// TIA Portal project "Factory IO Linha Completa" (V18)

(* hardware
DEVICE "S7-1500/ET200MP station_1"  S7-1500 station
   slot 0: "Rail_0"  Rack  6ES7 590-1***0-0AA0
   slot 1: "PLC_1"  CPU 1515-2 PN  6ES7 515-2AM00-0AB0  V1.8
      slot 3: "CPU display_1"  6ES7591-1BA00-0AA0
      slot 32768: "PROFINET interface_1"  X1
         slot 32769: "Port_1"  X1 P1
         slot 32770: "Port_2"  X1 P2
      slot 33024: "PROFINET interface_2"  X2
         slot 33025: "Port_1"  X2 P1
*)

// ===== PLC "PLC_1"  CPU 1515-2 PN =====

VAR_GLOBAL   // PLC tag table "Default tag table"
   "System_Byte" AT %MB1 : Byte;
   "FirstScan" AT %M1.0 : Bool;
   "DiagStatusUpdate" AT %M1.1 : Bool;
   "AlwaysTRUE" AT %M1.2 : Bool;
   "AlwaysFALSE" AT %M1.3 : Bool;
   "Clock_Byte" AT %MB0 : Byte;
   "Clock_10Hz" AT %M0.0 : Bool;
   "Clock_5Hz" AT %M0.1 : Bool;
   "Clock_2.5Hz" AT %M0.2 : Bool;
   "Clock_2Hz" AT %M0.3 : Bool;
   "Clock_1.25Hz" AT %M0.4 : Bool;
   "Clock_1Hz" AT %M0.5 : Bool;
   "Clock_0.625Hz" AT %M0.6 : Bool;
   "Clock_0.5Hz" AT %M0.7 : Bool;
END_VAR

VAR_GLOBAL   // PLC tag table "FactoryIO"
   "Emergency Stop 0" AT %I0.0 : Bool;
   "Start Button 0" AT %I0.1 : Bool;
   "Stop Button 0" AT %I0.2 : Bool;
   "Reset Button 0" AT %I0.3 : Bool;
   "Machining Center 0 (Is Busy)" AT %I0.5 : Bool;
   "Machining Center 0 (Has Error)" AT %I0.6 : Bool;
   "Machining Center 1 (Is Busy)" AT %I0.7 : Bool;
   "Machining Center 1 (Has Error)" AT %I1.0 : Bool;
   "Sensor 120" AT %I1.1 : Bool;
   "Sensor 122" AT %I1.2 : Bool;
   "Zne01 Conveyor 101" AT %Q0.0 : Bool;
   "Zne01 Conveyor 120" AT %Q0.1 : Bool;
   "Zne01 Conveyor 121" AT %Q0.2 : Bool;
   "Zne01 Conveyor 122" AT %Q0.3 : Bool;
   "Zne01 Conveyor 124" AT %Q0.4 : Bool;
   "Zne01 Conveyor 125" AT %Q0.5 : Bool;
   "Zne01 Sorter 102 (Up)" AT %Q0.6 : Bool;
   "Zne01 Sorter 102 (Left)" AT %Q0.7 : Bool;
   "Zne01 Sorter 102 (Right)" AT %Q1.0 : Bool;
   "Zne01 Sorter 123 (Up)" AT %Q1.1 : Bool;
   "Zne01 Sorter 123 (Right)" AT %Q1.2 : Bool;
   "Machining Center 0 (Start)" AT %Q1.3 : Bool;
   "Machining Center 0 (Stop)" AT %Q1.4 : Bool;
   "Machining Center 0 (Reset)" AT %Q1.5 : Bool;
   "Machining Center 1 (Start)" AT %Q1.6 : Bool;
   "Machining Center 1 (Stop)" AT %Q1.7 : Bool;
   "Machining Center 1 (Reset)" AT %Q2.0 : Bool;
   "Start Button 0 (Light)" AT %Q2.1 : Bool;
   "Stop Button 0 (Light)" AT %Q2.2 : Bool;
   "Reset Button 0 (Light)" AT %Q2.3 : Bool;
   "Vision Sensor 0 (Value)" AT %IW256 : Int;
   "Auto Selector 0" AT %I0.4 : Bool;
   "Machining Center 2 (Is Busy)" AT %I1.3 : Bool;
   "Machining Center 2 (Has Error)" AT %I1.4 : Bool;
   "Machining Center 3 (Is Busy)" AT %I1.5 : Bool;
   "Machining Center 3 (Has Error)" AT %I1.6 : Bool;
   "Sensor 130" AT %I1.7 : Bool;
   "Sensor 132" AT %I2.0 : Bool;
   "Zne01 Conveyor 130" AT %Q2.4 : Bool;
   "Zne01 Conveyor 131" AT %Q2.5 : Bool;
   "Zne01 Conveyor 132" AT %Q2.6 : Bool;
   "Zne01 Conveyor 134" AT %Q2.7 : Bool;
   "Zne01 Conveyor 135" AT %Q3.0 : Bool;
   "Zne01 Sorter 133 (Up)" AT %Q3.1 : Bool;
   "Zne01 Sorter 133 (Left)" AT %Q3.2 : Bool;
   "Machining Center 2 (Start)" AT %Q3.3 : Bool;
   "Machining Center 2 (Stop)" AT %Q3.4 : Bool;
   "Machining Center 2 (Reset)" AT %Q3.5 : Bool;
   "Machining Center 3 (Start)" AT %Q3.6 : Bool;
   "Machining Center 3 (Stop)" AT %Q3.7 : Bool;
   "Machining Center 3 (Reset)" AT %Q4.0 : Bool;
   "Zne02 Conveyor 220" AT %Q4.1 : Bool;
   "Zne02 Conveyor 221" AT %Q4.2 : Bool;
   "Zne02 Conveyor 222A" AT %Q4.3 : Bool;
   "Zne02 Conveyor 222B" AT %Q4.4 : Bool;
   "Zne02 Conveyor 223" AT %Q4.5 : Bool;
   "Zne02 Conveyor 224" AT %Q4.6 : Bool;
   "Zne02 Conveyor 225" AT %Q4.7 : Bool;
   "Zne03 Conveyor 300" AT %Q5.3 : Bool;
   "Zne03 Conveyor 301" AT %Q5.4 : Bool;
   "Zne03 Conveyor 302" AT %Q5.5 : Bool;
   "Sensor 223" AT %I2.1 : Bool;
   "Sensor 225" AT %I2.2 : Bool;
   "Zne02 Clamp Closed" AT %I2.3 : Bool;
   "Zne02 Clamp Limit" AT %I2.4 : Bool;
   "Zne02 Pusher" AT %Q5.0 : Bool;
   "Zne02 Clamp" AT %Q5.1 : Bool;
   "Zne02 Clamp Rise" AT %Q5.2 : Bool;
   "Vision Sensor 2 (Value)" AT %IW258 : Int;
   "Sensor 300" AT %I2.5 : Bool;
   "Sensor 301" AT %I2.6 : Bool;
   "Sensor 302" AT %I2.7 : Bool;
   "Zne03 (Detected)" AT %I3.0 : Bool;
   "Zne03 (Moving X)" AT %I3.1 : Bool;
   "Zne03 (Moving Z)" AT %I3.2 : Bool;
   "Zne03 Clamp Closed" AT %I3.3 : Bool;
   "Zne03 Clamp Limit" AT %I3.4 : Bool;
   "Zne03 Clamp" AT %Q5.6 : Bool;
   "Zne03 Clamp Raise" AT %Q5.7 : Bool;
   "Zne03 X" AT %Q6.0 : Bool;
   "Zne03 Z" AT %Q6.1 : Bool;
   "Zne03 (Grab)" AT %Q6.2 : Bool;
   "Zne03 Pusher" AT %Q6.3 : Bool;
   "Vision Sensor 1 (Value)" AT %IW260 : Int;
   "Sensor 423" AT %I3.5 : Bool;
   "Sensor 425" AT %I3.6 : Bool;
   "Zne04 Clamp Closed" AT %I3.7 : Bool;
   "Zne04 Clamp Limit" AT %I4.0 : Bool;
   "Sensor 500" AT %I4.1 : Bool;
   "Sensor 501" AT %I4.2 : Bool;
   "Sensor 502" AT %I4.3 : Bool;
   "Zne05 (Detected)" AT %I4.4 : Bool;
   "Zne05 (Moving X)" AT %I4.5 : Bool;
   "Zne05 (Moving Z)" AT %I4.6 : Bool;
   "Zne05 Clamp Closed" AT %I4.7 : Bool;
   "Zne05 Clamp Limit" AT %I5.0 : Bool;
   "Zne04 Conveyor 420" AT %Q6.4 : Bool;
   "Zne04 Conveyor 421" AT %Q6.5 : Bool;
   "Zne04 Conveyor 422B" AT %Q6.7 : Bool;
   "Zne04 Conveyor 423" AT %Q7.0 : Bool;
   "Zne04 Conveyor 424" AT %Q7.1 : Bool;
   "Zne04 Conveyor 425" AT %Q7.2 : Bool;
   "Zne04 Pusher" AT %Q7.3 : Bool;
   "Zne04 Clamp" AT %Q7.4 : Bool;
   "Zne04 Clamp Raise" AT %Q7.5 : Bool;
   "Zne05 Conveyor 500" AT %Q7.6 : Bool;
   "Zne05 Conveyor 501" AT %Q7.7 : Bool;
   "Zne05 Conveyor 502" AT %Q8.0 : Bool;
   "Zne05 Clamp" AT %Q8.1 : Bool;
   "Zne05 Clamp Raise" AT %Q8.2 : Bool;
   "Zne05 X" AT %Q8.3 : Bool;
   "Zne05 Z" AT %Q8.4 : Bool;
   "Zne05 (Grab)" AT %Q8.5 : Bool;
   "Zne05 Pusher" AT %Q8.6 : Bool;
   "Vision Sensor 3 (Value)" AT %IW262 : Int;
   "Vision Sensor 4 (Value)" AT %IW264 : Int;
   "Zne04 Conveyor 422A" AT %Q6.6 : Bool;
   "Sensor 920" AT %I10.0 : Bool;
   "Sensor 921" AT %I10.1 : Bool;
   "Sensor 922" AT %I10.2 : Bool;
   "Sensor 930" AT %I10.3 : Bool;
   "Sensor 931" AT %I10.4 : Bool;
   "Sensor 932" AT %I10.5 : Bool;
   "Sensor 950" AT %I10.6 : Bool;
   "Sensor 951" AT %I10.7 : Bool;
   "Sensor 952" AT %I11.0 : Bool;
   "Sensor 953" AT %I11.1 : Bool;
   "Zne09 Conveyor 920" AT %Q10.0 : Bool;
   "Zne09 Conveyor 921" AT %Q10.1 : Bool;
   "Zne09 Conveyor 930" AT %Q10.2 : Bool;
   "Zne09 Conveyor 931" AT %Q10.3 : Bool;
   "Zne09 Conveyor 950" AT %Q10.4 : Bool;
   "Zne09 Conveyor 951" AT %Q10.5 : Bool;
   "Zne09 Conveyor 952" AT %Q10.6 : Bool;
   "Zne09 Conveyor 953" AT %Q10.7 : Bool;
   "Zne09 Chain Transfer Right" AT %Q11.0 : Bool;
   "Zne09 Chain Transfer Left" AT %Q11.1 : Bool;
   "Zne09 Chain Transfer Foward" AT %Q11.2 : Bool;
   "Zne09 Chain Transfer Backward" AT %Q11.3 : Bool;
   "Pick & Place 0 X Position (V)" AT %IW266 : Int;
   "Pick & Place 0 Y Position (V)" AT %IW268 : Int;
   "Pick & Place 0 Z Position (V)" AT %IW270 : Int;
   "Pick & Place 1 X Position (V)" AT %IW272 : Int;
   "Pick & Place 1 Y Position (V)" AT %IW274 : Int;
   "Pick & Place 1 Z Position (V)" AT %IW276 : Int;
   "Pick & Place 0 X Set Point (V)" AT %QW256 : Int;
   "Pick & Place 0 Y Set Point(V)" AT %QW258 : Int;
   "Pick & Place 0 Z Set Point (V)" AT %QW260 : Int;
   "Pick & Place 1 X Set Point (V)" AT %QW262 : Int;
   "Pick & Place 1 Y Set Point(V)" AT %QW264 : Int;
   "Pick & Place 1 Z Set Point (V)" AT %QW266 : Int;
   "Zne09 Stacker Target Position" AT %QW270 : Int;
   "Pick & Place 1 (Box Detected)" AT %I11.2 : Bool;
   "Pick & Place 0 (Box Detected)" AT %I11.3 : Bool;
   "Pick & Place 1 (Grab)" AT %Q11.4 : Bool;
   "Pick & Place 0 (Grab)" AT %Q11.5 : Bool;
   "AtRight" AT %I12.0 : Bool;
   "AtLeft" AT %I12.1 : Bool;
   "AtCenter" AT %I12.2 : Bool;
   "MovingX" AT %I12.3 : Bool;
   "MovingZ" AT %I12.4 : Bool;
   "Forks RIght" AT %Q12.0 : Bool;
   "ForksLeft" AT %Q12.1 : Bool;
   "Lift" AT %Q12.2 : Bool;
END_VAR

VAR_GLOBAL CONSTANT   // PLC tag table "FactoryIO"
   "BlueRawMaterial" : Int := 1;
   "GreenRawMaterial" : Int := 4;
   "HOMEPOSITION" : Int := 255;
   "BlueLidMaterial" : Int := 2;
   "GreenLidMaterial" : Int := 5;
   "BlueBaseMaterial" : Int := 3;
   "GreenBaseMaterial" : Int := 6;
   "MaxCoordinates" : Int := 10;
END_VAR

TYPE "St_Conveyor"
   STRUCT
      IHM_xButtonRun : Bool;
      IHM_xStatusMotor : Int;
      iq_xError : Bool;
      iq_iErrorType : Int;
   END_STRUCT;
END_TYPE

TYPE "St_ControlPanel"
   STRUCT
      q_xManualMode : Bool;
      q_xAutoMode : Bool;
      q_xEmergencyStatusZone : Bool;
      q_xPanelResetCmd : Bool;
      iq_xPanelOn : Bool;
      iq_xPanelOff : Bool;
      iq_xError : Bool;
      iq_iErrorType : Int;
      q_siMode : Int;
      iq_sFaultDescription : String;
   END_STRUCT;
END_TYPE

TYPE "St_Warehouse"
   STRUCT
      xPedidoRetirada : Bool;
      xFimMovimento : Bool;
      xPosiçaoLivre : Bool;
      iPosição : Int;
      xSensorEntrada : Bool;
      xSensorSaida : Bool;
      iMachineState_Entrada : Int;
      iMachineState_Retirada : Int;
      xForksLeft : Bool;
      xForksRight : Bool;
      xLift : Bool;
      q_dTargetPosition : DInt;
      Armazem : Array[1..54] of Bool;
      iStateRetirada : String;
      iStateEntrada : String;
   END_STRUCT;
END_TYPE

TYPE "St_Sorter"
   STRUCT
      temp : Bool;
   END_STRUCT;
END_TYPE

TYPE "St_Assembler"
   STRUCT
      LidClampUpPosition : Bool;
      LidClampDownPosition : Bool;
      BaseClampUpPosition : Bool;
      BaseClampDownPosition : Bool;
      AxisXFoward : Bool;
      AxisXBackward : Bool;
      AxisZRise : Bool;
      AxisZDown : Bool;
      iMachineState : Int;
      iState : String;
      MemoryPresenceLid : Bool;
      MemoryPresenceBase : Bool;
      ReadyToReceiveLid : Bool;
      ReadyToReceiveBase : Bool;
      EnableSend : Bool;
   END_STRUCT;
END_TYPE

TYPE "St_Manipulator"
   STRUCT
      ReadyToReceivePallet : Bool;
      PalletFull : Bool;
      ContActual : Int;
      ContMax : Int;
      iMachineState : Int;
      iState : String;
      Coordinates : Array[0.."MaxCoordinates"] of Struct
         "Axis X" : Int;
         "Axis Y" : Int;
         "Axis Z" : Int;
      END_STRUCT;
      Ack_Positions : Array[0.."MaxCoordinates"] of Bool;
   END_STRUCT;
END_TYPE

TYPE "St_Transfer"
   STRUCT
      EnableSend : Bool;
      RequestRight : Bool;
      RequestLeft : Bool;
      ReadyToReceiveRight : Bool;
      ReadyToReceiveLeft : Bool;
      LastReceiveRightSide : Bool;
      "Chain Transfer Foward" : Bool;
      "Chain Transfer Backward" : Bool;
      "Chain Transfer Right" : Bool;
      "Chain Transfer Left" : Bool;
      iMachineState : Int;
      iState : String;
   END_STRUCT;
END_TYPE

DATA_BLOCK "General"   // DB2
{ S7_Optimized_Access := 'TRUE' }
VERSION : 0.1
   VAR
      Panel01 : "St_ControlPanel";
      "Conveyor 101" : "St_Conveyor";
      "Conveyor 120" : "St_Conveyor";
      "Conveyor 121" : "St_Conveyor";
      "Conveyor 122" : "St_Conveyor";
      "Conveyor 124" : "St_Conveyor";
      "Conveyor 125" : "St_Conveyor";
      "Conveyor 130" : "St_Conveyor";
      "Conveyor 131" : "St_Conveyor";
      "Conveyor 132" : "St_Conveyor";
      "Conveyor 134" : "St_Conveyor";
      "Conveyor 135" : "St_Conveyor";
      "Conveyor 220" : "St_Conveyor";
      "Conveyor 221" : "St_Conveyor";
      "Conveyor 222" : "St_Conveyor";
      "Conveyor 223" : "St_Conveyor";
      "Conveyor 224" : "St_Conveyor";
      "Conveyor 225" : "St_Conveyor";
      "Conveyor 300" : "St_Conveyor";
      "Conveyor 301" : "St_Conveyor";
      "Conveyor 302" : "St_Conveyor";
      "Assembler Zne03" : "St_Assembler";
      "Conveyor 420" : "St_Conveyor";
      "Conveyor 421" : "St_Conveyor";
      "Conveyor 422" : "St_Conveyor";
      "Conveyor 423" : "St_Conveyor";
      "Conveyor 424" : "St_Conveyor";
      "Conveyor 425" : "St_Conveyor";
      "Conveyor 500" : "St_Conveyor";
      "Conveyor 501" : "St_Conveyor";
      "Conveyor 502" : "St_Conveyor";
      "Assembler Zne05" : "St_Assembler";
      "Conveyor 920" : "St_Conveyor";
      "Conveyor 921" : "St_Conveyor";
      "Manipulator 1" : "St_Manipulator";
      "Conveyor 930" : "St_Conveyor";
      "Conveyor 931" : "St_Conveyor";
      "Manipulator 0" : "St_Manipulator";
      Transfer : "St_Transfer";
      "Conveyor 950" : "St_Conveyor";
      "Conveyor 951" : "St_Conveyor";
      Warehouse : "St_Warehouse";
      "Conveyor 952" : "St_Conveyor";
      "Conveyor 953" : "St_Conveyor";
   END_VAR
BEGIN
END_DATA_BLOCK

// folder: PANEL

DATA_BLOCK "ControlPanel_DB"   // DB1
{ S7_Optimized_Access := 'TRUE' }
VERSION : 0.1
// stored: InstanceOfName ControlPanel
"ControlPanel"
BEGIN
END_DATA_BLOCK

// folder: ZNE01

DATA_BLOCK "Zne01_DB"   // DB3
{ S7_Optimized_Access := 'TRUE' }
VERSION : 0.1
// stored: InstanceOfName Zne01
"Zne01"
BEGIN
END_DATA_BLOCK

// folder: ZNE02

DATA_BLOCK "Zne02_DB"   // DB4
{ S7_Optimized_Access := 'TRUE' }
VERSION : 0.1
// stored: InstanceOfName Zne02
"Zne02"
BEGIN
END_DATA_BLOCK

// folder: ZNE03

DATA_BLOCK "Zne03_DB"   // DB5
{ S7_Optimized_Access := 'TRUE' }
VERSION : 0.1
// stored: InstanceOfName Zne03
"Zne03"
BEGIN
END_DATA_BLOCK

// folder: ZNE04

DATA_BLOCK "Zne04_DB"   // DB6
{ S7_Optimized_Access := 'TRUE' }
VERSION : 0.1
// stored: InstanceOfName Zne04
"Zne04"
BEGIN
END_DATA_BLOCK

// folder: ZNE05

DATA_BLOCK "Zne05_DB"   // DB7
{ S7_Optimized_Access := 'TRUE' }
VERSION : 0.1
// stored: InstanceOfName Zne05
"Zne05"
BEGIN
END_DATA_BLOCK

// folder: ZNE09

DATA_BLOCK "Zne09_DB"   // DB8
{ S7_Optimized_Access := 'TRUE' }
VERSION : 0.1
// stored: InstanceOfName Zne09
"Zne09"
BEGIN
END_DATA_BLOCK

// folder: (top level)

ORGANIZATION_BLOCK "Main_1"   // OB123, SCL, ProgramCycle
TITLE = "Main Program Sweep (Cycle)"
{ S7_Optimized_Access := 'TRUE' }
VERSION : 0.1
   VAR_INPUT
      Initial_Call : Bool;   // Initial call of this OB
      Remanence : Bool;   // =True, if remanent data are available
   END_VAR
BEGIN


   "MHJ-PLC-Lab-Function-S71200"();

   "ControlPanel_DB"(i_xButtonReset:="Reset Button 0",
                     i_xButtonStart:="Start Button 0",
                     i_xButtonStop:="Stop Button 0",
                     i_xButtonEmergency:="Emergency Stop 0",
                     i_xSelectorMode:="Auto Selector 0",
                     i_xClock:="Clock_1Hz",
                     q_xStartLight=>"Start Button 0 (Light)",
                     q_xStopLight=>"Stop Button 0 (Light)",
                     q_xResetLight=>"Reset Button 0 (Light)",
                     ControlPanel:="General".Panel01);

   "Zne01_DB"(); 
   "Zne02_DB"();
   "Zne03_DB"();
   "Zne04_DB"();
   "Zne05_DB"();
   "Receita"();
   "Zne09_DB"();
END_ORGANIZATION_BLOCK

// folder: PANEL

FUNCTION_BLOCK "ControlPanel"   // FB1, SCL
{ S7_Optimized_Access := 'TRUE' }
VERSION : 0.1
   VAR_INPUT
      i_xButtonReset : Bool;
      i_xButtonStart : Bool;
      i_xButtonStop : Bool;
      i_xButtonEmergency : Bool;
      i_xSelectorMode : Bool;   // 0 = Manual, 1= Auto
      i_xClock : Bool;
   END_VAR
   VAR_OUTPUT
      q_xStartLight : Bool;
      q_xStopLight : Bool;
      q_xResetLight : Bool;
   END_VAR
   VAR_IN_OUT
      ControlPanel : "St_ControlPanel";
   END_VAR
   VAR
      IEC_Timer_0_Instance : TON_TIME;
   END_VAR
BEGIN
   REGION INPUTS
       //EMERGENCY STATUS//
       IF #i_xButtonEmergency AND #i_xButtonReset THEN
           #ControlPanel.q_xEmergencyStatusZone := TRUE;
       ELSIF NOT #i_xButtonEmergency THEN
           #ControlPanel.q_xEmergencyStatusZone := FALSE;
       END_IF;

       //MANUAL MODE//
       IF #ControlPanel.q_xEmergencyStatusZone AND NOT #i_xSelectorMode THEN
           #ControlPanel.q_xManualMode := TRUE;
       ELSIF NOT #ControlPanel.q_xEmergencyStatusZone OR #i_xSelectorMode THEN
           #ControlPanel.q_xManualMode := FALSE;
       END_IF;

       //AUTO MODE//
       IF #ControlPanel.q_xEmergencyStatusZone AND #i_xSelectorMode AND #ControlPanel.iq_xPanelOn THEN
           #ControlPanel.q_xAutoMode := TRUE;
       ELSIF NOT #ControlPanel.q_xEmergencyStatusZone OR NOT #i_xSelectorMode OR #ControlPanel.iq_xPanelOff THEN
           #ControlPanel.q_xAutoMode := FALSE;
       END_IF;

       //RESET COMMAND//
       #IEC_Timer_0_Instance(IN:=#i_xButtonReset,
                             PT:=t#5s,
                             Q=>#ControlPanel.q_xPanelResetCmd);

       //ON-OFF COMMAND//
       IF #i_xButtonStart AND #i_xButtonStop THEN
           #ControlPanel.iq_xPanelOn := TRUE;
           #ControlPanel.iq_xPanelOff := FALSE;
       ELSIF NOT #i_xButtonStop OR NOT #ControlPanel.q_xEmergencyStatusZone OR #ControlPanel.q_xManualMode THEN
           #ControlPanel.iq_xPanelOn := FALSE;
           #ControlPanel.iq_xPanelOff := TRUE;
       END_IF;
   END_REGION

   REGION STATUS MODE
       IF NOT #ControlPanel.q_xEmergencyStatusZone THEN
           #ControlPanel.q_siMode := 1; //EMERGENCIA

       ELSIF #ControlPanel.q_xAutoMode THEN
           #ControlPanel.q_siMode := 2; //AUTOMATICO

       ELSIF #ControlPanel.q_xManualMode THEN
           #ControlPanel.q_siMode := 3; //MANUAL

       ELSE
           #ControlPanel.q_siMode := 4; //DESLIGADO
       END_IF;
   END_REGION

   REGION OUTPUTS
       //START LIGHT    
       #q_xStartLight := #ControlPanel.q_xAutoMode OR (#i_xSelectorMode AND #ControlPanel.q_xEmergencyStatusZone AND #i_xClock);
       //STOP LIGHT 
       #q_xStopLight := NOT #i_xButtonEmergency OR (#i_xButtonEmergency AND NOT #ControlPanel.q_xEmergencyStatusZone AND #i_xClock);
       //RESET LIGHT 
       #q_xResetLight := #ControlPanel.q_xPanelResetCmd;
   END_REGION
END_FUNCTION_BLOCK

// folder: STANDARD BLOCKS

FUNCTION_BLOCK "Conveyor"   // FB2, SCL
{ S7_Optimized_Access := 'TRUE' }
VERSION : 0.1
   VAR_INPUT
      i_xInterlock : Bool;
      i_xRun : Bool;
      ControlPanel : "St_ControlPanel";
   END_VAR
   VAR_OUTPUT
      q_xMotorOn : Bool := false;
   END_VAR
   VAR_IN_OUT
      Conveyor : "St_Conveyor";
   END_VAR
BEGIN

   REGION MODO
       CASE #ControlPanel.q_siMode OF
           1:  // EMERGENCIA
               #q_xMotorOn := FALSE;

           2:  // AUTOMATICO
               IF #i_xRun AND NOT #i_xInterlock THEN
                   #q_xMotorOn := TRUE;
               ELSE
                   #q_xMotorOn := FALSE;
               END_IF;

           3:  // MANUAL
               #q_xMotorOn := #Conveyor.IHM_xButtonRun;

           ELSE
               #q_xMotorOn := FALSE;
       END_CASE;
   END_REGION

   REGION #IHM
       IF #Conveyor.iq_xError THEN
           #Conveyor.IHM_xStatusMotor := 1; // ERRO

       ELSIF #ControlPanel.q_xAutoMode AND #q_xMotorOn THEN
           #Conveyor.IHM_xStatusMotor := 2; // AUTO RUNNING

       ELSIF #ControlPanel.q_xManualMode AND #q_xMotorOn THEN
           #Conveyor.IHM_xStatusMotor := 3; // MANUAL RUNNING

       ELSIF NOT #q_xMotorOn THEN
           #Conveyor.IHM_xStatusMotor := 4; // MOTOR STOPED

       END_IF;
   END_REGION
END_FUNCTION_BLOCK

FUNCTION_BLOCK "Warehouse"   // FB3, SCL
{ S7_Optimized_Access := 'TRUE' }
VERSION : 0.1
   VAR_INPUT
      i_xAtLeft : Bool;
      i_xAtRight : Bool;
      i_xAtMiddle : Bool;
      i_xMovingZ : Bool;
      i_xMovingX : Bool;
      ControlPanel : "St_ControlPanel";
   END_VAR
   VAR_OUTPUT
      q_xForksLeft : Bool;
      q_xForksRight : Bool;
      q_xLift : Bool;
      q_dTargetPosition : Int;
   END_VAR
   VAR_IN_OUT
      Warehouse : "St_Warehouse";
   END_VAR
   VAR
      t_LiftDown : TON_TIME;
      t_LiftUp : TON_TIME;
      TargetPositionRetirada : DInt;
      TargetPositionEntrada : DInt;
      t_NotMovingX : TON_TIME;
   END_VAR
BEGIN

   IF #ControlPanel.q_xPanelResetCmd THEN
       #Warehouse.xForksLeft := 0;
       #Warehouse.xForksRight := 0;
       #Warehouse.xLift := 0;
       #Warehouse.q_dTargetPosition := "HOMEPOSITION";
       #Warehouse.iMachineState_Entrada := 0;
       #Warehouse.iMachineState_Retirada := 0;
       #Warehouse.iPosição := 0;
   END_IF;


   IF #Warehouse.iPosição > 54 THEN
       #Warehouse.iPosição := 54;
   END_IF;

   IF #Warehouse.iPosição < 1 THEN
       #Warehouse.iPosição := 1;
   END_IF;

   REGION TIMMERS
       #t_LiftDown(IN := NOT #q_xLift AND NOT #i_xMovingZ,
                   PT := T#1s);

       #t_LiftUp(IN:=#q_xLift AND NOT #i_xMovingZ,
                 PT:=T#1s);

       #t_NotMovingX(IN:= NOT #i_xMovingX,
                  PT:=T#2s);
   END_REGION

   REGION ESTADO RETIRADA
       IF #ControlPanel.q_xAutoMode AND #Warehouse.iMachineState_Entrada <= 1 THEN

           CASE #Warehouse.iMachineState_Retirada OF
               0:  // AGUARDANDO SOLICITAÇÃO RETIRADA
                   #Warehouse.iStateRetirada := 'S00 - AGUARDANDO SOLICITACAO RETIRADA';
                   IF #Warehouse.xPedidoRetirada THEN
                       #Warehouse.iMachineState_Retirada := 1;
                   END_IF;

               1:  // VERIFICA POSICAO VALIDA
                   #Warehouse.iStateRetirada := 'S01 - VERIFICA POSICAO VALIDA';
                   IF #Warehouse.Armazem[#Warehouse.iPosição] THEN
                       #Warehouse.iMachineState_Retirada := 3;
                       #TargetPositionRetirada := #Warehouse.iPosição;
                   ELSE
                       #Warehouse.iMachineState_Retirada := 2;
                   END_IF;

               2:  // POSICAO INVALIDA
                   #Warehouse.iStateRetirada := 'S02 - POSICAO INVALIDA PARA RETIRADA';
                   IF NOT #Warehouse.xPedidoRetirada THEN
                       #Warehouse.iMachineState_Retirada := 0;
                   END_IF;

               3:  // FORK LIVRE
                   #Warehouse.iStateRetirada := 'S03 - REPOUSO FORKS';
                   #Warehouse.xLift := 0;
                   IF #t_LiftDown.Q THEN
                       #Warehouse.xForksLeft := 0;
                       #Warehouse.xForksRight := 0;
                       IF #i_xAtMiddle THEN
                           #Warehouse.iMachineState_Retirada := 4;
                       END_IF;
                   END_IF;

               4:  // DESLOCA PARA POSICAO DO ARMAZEM
                   #Warehouse.iStateRetirada := 'S04 - DESLOCA PARA POSICAO DO ARMAZEM';
                   #Warehouse.q_dTargetPosition := #TargetPositionRetirada;
                   IF (#q_dTargetPosition = #Warehouse.q_dTargetPosition) AND #t_NotMovingX.Q THEN
                       #Warehouse.iMachineState_Retirada := 5;
                   END_IF;

               5:  // AVANCA FORK
                   #Warehouse.iStateRetirada := 'S05 - AVANCA FORK';
                   #Warehouse.xForksRight := 1;
                   IF #q_xForksRight AND #i_xAtRight THEN
                       #Warehouse.iMachineState_Retirada := 6;
                   END_IF;

               6:  // LIFT UP
                   #Warehouse.iStateRetirada := 'S06 - ERGUE LIFT';
                   #Warehouse.xLift := 1;
                   IF #q_xLift AND #t_LiftUp.Q THEN
                       #Warehouse.Armazem[#TargetPositionRetirada] := 0;
                       IF NOT #Warehouse.Armazem[#TargetPositionRetirada] THEN
                           #Warehouse.iMachineState_Retirada := 7;
                       END_IF;
                   END_IF;

               7:  // RECUA FORKS
                   #Warehouse.iStateRetirada := 'S07 - RECUA FORKS';
                   #Warehouse.xForksRight := 0;
                   IF NOT #q_xForksRight AND #i_xAtMiddle THEN
                       #Warehouse.iMachineState_Retirada := 8;
                   END_IF;

               8:  // DESLOCA PARA POSICAO DAS ESTEIRA DE SAIDA
                   #Warehouse.iStateRetirada := 'S08 - DESLOCA PARA POSICAO DAS ESTEIRA DE SAIDA';
                   #Warehouse.q_dTargetPosition := "HOMEPOSITION";
                   IF #t_NotMovingX.Q AND (#q_dTargetPosition = "HOMEPOSITION") AND NOT #Warehouse.xSensorSaida THEN
                       #Warehouse.iMachineState_Retirada := 9;
                   END_IF;

               9:  // AVANCA FORK PARA ENVIO ESTEIRA
                   #Warehouse.iStateRetirada := 'S09 - AVANCA FORK PARA ENVIO ESTEIRA';
                   #Warehouse.xForksRight := 1;
                   IF #q_xForksRight AND #i_xAtRight THEN
                       #Warehouse.iMachineState_Retirada := 10;
                   END_IF;

               10: // LIFT DOWN
                   #Warehouse.iStateRetirada := 'S10 - DEPOSITA PALLET NA ESTEIRA';
                   #Warehouse.xLift := 0;
                   IF NOT #q_xLift AND #t_LiftDown.Q THEN
                       #Warehouse.iMachineState_Retirada := 11;
                   END_IF;

               11: // RECUA FORKS
                   #Warehouse.iStateRetirada := 'S11 - RECUA FORKS';
                   #Warehouse.xForksRight := 0;
                   IF NOT #q_xForksRight AND #i_xAtMiddle AND NOT #Warehouse.xPedidoRetirada THEN
                       #Warehouse.iMachineState_Retirada := 0;
                       #Warehouse.iStateRetirada := 'S00 - AGUARDANDO SOLICITACAO RETIRADA';
                   END_IF;

               ELSE
                   #Warehouse.iMachineState_Retirada := 0;
           END_CASE;
       END_IF;
   END_REGION

   REGION ESTADO DEPOSITO 

       IF #ControlPanel.q_xAutoMode AND #Warehouse.iMachineState_Retirada = 0 THEN

           CASE #Warehouse.iMachineState_Entrada OF

               0: //POSICAO LIVRE INDISPONIVEL
                   #Warehouse.iStateEntrada := 'S00 - POSICAO LIVRE INDISPONIVEL';
                   #TargetPositionEntrada := "PosDisponivel"(#Warehouse.Armazem);
                   IF #TargetPositionEntrada <> -1 THEN
                       #Warehouse.iMachineState_Entrada := 1;
                   END_IF;

               1:  // AGUARDANDO CHEGADA PALLET
                   #Warehouse.iStateEntrada := 'S01 - AGUARDANDO CHEGADA PALLET';
                   IF #Warehouse.xSensorEntrada AND NOT #Warehouse.xPedidoRetirada THEN
                       #Warehouse.iMachineState_Entrada := 2;
                   END_IF;

               2:   // VERIFICA POSICAO DISPONIVEL
                   #Warehouse.iStateEntrada := 'S02 - VERIFICA POSICAO DISPONIVEL';
                   #TargetPositionEntrada := "PosDisponivel"(#Warehouse.Armazem);
                   IF #TargetPositionEntrada = -1 THEN
                       #Warehouse.iMachineState_Entrada := 0;
                   ELSE
                       #Warehouse.iMachineState_Entrada := 3;
                   END_IF;

               3: // FORKS LIVRE
                   #Warehouse.iStateEntrada := 'S03 - REPOUSO FORKS';
                   #Warehouse.xLift := 0;
                   IF #t_LiftDown.Q THEN
                       #Warehouse.xForksLeft := 0;
                       #Warehouse.xForksRight := 0;
                       IF #i_xAtMiddle THEN
                           #Warehouse.iMachineState_Entrada := 4;
                       END_IF;
                   END_IF;

               4: // DESLOCA PARA POSICAO DA ESTEIRA DE ENTRADA
                   #Warehouse.iStateEntrada := 'S04 - DESLOCA PARA POSICAO DA ESTEIRA DE ENTRADA';
                   #Warehouse.q_dTargetPosition := "HOMEPOSITION";
                   IF #q_dTargetPosition = "HOMEPOSITION" AND #t_NotMovingX.Q THEN
                       #Warehouse.iMachineState_Entrada := 5;
                   END_IF;

               5: // AVANÇA FORKS
                   #Warehouse.iStateEntrada := 'S05 - AVANCA FORKS';
                   #Warehouse.xForksLeft := 1;
                   IF #q_xForksLeft AND #i_xAtLeft THEN
                       #Warehouse.iMachineState_Entrada := 6;
                   END_IF;

               6:  // RETIRAR PALLET
                   #Warehouse.iStateEntrada := 'S06 - RETIRAR PALLET';
                   #Warehouse.xLift := 1;
                   IF #q_xLift AND #t_LiftUp.Q AND NOT #Warehouse.xSensorEntrada THEN
                       #Warehouse.iMachineState_Entrada := 7;
                   END_IF;

               7: // RECUA FORKS
                   #Warehouse.iStateEntrada := 'S07 - RECUA FORKS';
                   #Warehouse.xForksLeft := 0;
                   IF NOT #Warehouse.xForksLeft AND #i_xAtMiddle THEN
                       #Warehouse.iMachineState_Entrada := 8;
                   END_IF;

               8: // DESLOCA PARA POSICAO DE DEPOSITO NO ARMAZEM
                   #Warehouse.iStateEntrada := 'S08 - DESLOCA PARA POSICAO DE DEPOSITO NO ARMAZEM';
                   #Warehouse.q_dTargetPosition := #TargetPositionEntrada;
                   IF #q_dTargetPosition = #TargetPositionEntrada AND #t_NotMovingX.Q THEN
                       #Warehouse.iMachineState_Entrada := 9;
                   END_IF;

               9: // AVANÇA FORKS NO ARMAZEM
                   #Warehouse.iStateEntrada := 'S09 - AVANCA FORKS NO ARMAZEM';
                   #Warehouse.xForksRight := 1;
                   IF #q_xForksRight AND #i_xAtRight THEN
                       #Warehouse.iMachineState_Entrada := 10;
                   END_IF;

               10: // DEPOSITA PALLET
                   #Warehouse.iStateEntrada := 'S10 - DEPOSITA PALLET';
                   #Warehouse.xLift := 0;
                   IF NOT #q_xLift AND #t_LiftDown.Q THEN
                       #Warehouse.Armazem[#q_dTargetPosition] := 1;
                       #Warehouse.iMachineState_Entrada := 11;
                   END_IF;

               11: // RECUA FORKS
                   #Warehouse.iStateEntrada := 'S11 - RECUA FORKS APOS DEPOSITO';
                   #Warehouse.xForksRight := 0;
                   IF NOT #q_xForksRight AND #i_xAtMiddle THEN
                       #Warehouse.iMachineState_Entrada := 0;
                   END_IF;

               ELSE  
                   #Warehouse.iMachineState_Entrada := 0;
           END_CASE;
       END_IF;
   END_REGION




   REGION OUTPUTS
       IF #ControlPanel.q_xAutoMode THEN

           IF #t_NotMovingX.Q THEN 
               #q_xForksLeft := #Warehouse.xForksLeft;
               #q_xForksRight := #Warehouse.xForksRight;
               #q_xLift := #Warehouse.xLift;
           END_IF;

           IF #i_xAtMiddle AND NOT #q_xForksLeft AND NOT #q_xForksRight THEN 
               #q_dTargetPosition := #Warehouse.q_dTargetPosition;
           END_IF;

       END_IF;
   END_REGION
END_FUNCTION_BLOCK

FUNCTION_BLOCK "Sorter"   // FB5, SCL
{ S7_Optimized_Access := 'TRUE' }
VERSION : 0.1
   VAR_INPUT
      i_xRightRequest : Bool;
      i_xLeftRequest : Bool;
      i_xCenterRequest : Bool;
      ControlPanel : "St_ControlPanel";
   END_VAR
   VAR_OUTPUT
      q_xUp : Bool;
      q_xRight : Bool;
      q_xLeft : Bool;
   END_VAR
BEGIN

   REGION MODO
       CASE #ControlPanel.q_siMode OF
           1:  // EMERGENCIA
               #q_xUp := FALSE;

           2:  // AUTOMATICO
               #q_xUp := TRUE;

               IF #i_xRightRequest THEN
                   #q_xRight := TRUE;
                   #q_xLeft := FALSE;
               END_IF;

               IF #i_xLeftRequest THEN
                   #q_xRight := FALSE;
                   #q_xLeft := TRUE;
               END_IF;

               IF #i_xCenterRequest THEN
                   #q_xRight := FALSE;
                   #q_xLeft := FALSE;
               END_IF;

           3:  // MANUAL
               #q_xUp := FALSE;

           ELSE
               #q_xUp := FALSE;
       END_CASE;
   END_REGION
END_FUNCTION_BLOCK

FUNCTION_BLOCK "MachineCenter"   // FB6, SCL
{ S7_Optimized_Access := 'TRUE' }
VERSION : 0.1
   VAR_INPUT
      Interlock : Bool;
      ControlPanel : "St_ControlPanel";
   END_VAR
   VAR_OUTPUT
      Start : Bool;
      Stop : Bool;
      Reset : Bool;
   END_VAR
BEGIN
   REGION MODO
       CASE #ControlPanel.q_siMode OF
           1:  // EMERGENCIA
               #Start := FALSE;
               #Stop := TRUE;

           2:  // AUTOMATICO
               IF NOT #Interlock THEN
                   #Start := TRUE;
                   #Stop := FALSE;
               ELSE
                   #Start := FALSE;
                   #Stop := TRUE;
               END_IF;

           3:  // MANUAL
               #Start := FALSE;
               #Stop := TRUE;

           ELSE
               #Start := FALSE;
               #Stop := TRUE;
       END_CASE;
   END_REGION

   #Reset := #ControlPanel.q_xPanelResetCmd;
END_FUNCTION_BLOCK

FUNCTION_BLOCK "Pusher"   // FB8, SCL
{ S7_Optimized_Access := 'TRUE' }
VERSION : 0.1
   VAR_INPUT
      RequestPusher : Bool;
      "Timer" : Time;
      ControlPanel : "St_ControlPanel";
   END_VAR
   VAR_OUTPUT
      Pusher : Bool;
   END_VAR
   VAR
      RequestPusherDelay : TON_TIME;
   END_VAR
BEGIN

   REGION MODO
       CASE #ControlPanel.q_siMode OF
           1:  // EMERGENCIA
               #Pusher := FALSE;

           2:  // AUTOMATICO
               #RequestPusherDelay(IN:=#RequestPusher,
                                   PT:=#Timer);

               IF #RequestPusherDelay.Q THEN
                   #Pusher := TRUE;
               ELSE
                   #Pusher := FALSE;
               END_IF;

           3:  // MANUAL
               #Pusher := FALSE;

           ELSE
               #Pusher := FALSE;
       END_CASE;
   END_REGION
END_FUNCTION_BLOCK

FUNCTION_BLOCK "Assembler"   // FB10, SCL
{ S7_Optimized_Access := 'TRUE' }
VERSION : 0.1
   VAR_INPUT
      LidClampClosed : Bool;
      LidClampLimit : Bool;
      BaseClampClosed : Bool;
      BaseClampLimit : Bool;
      PresenceLidConveyor : Bool;
      PresenceBaseConveyor : Bool;
      PresenceGrab : Bool;
      MovingX : Bool;
      MovingZ : Bool;
      ControlPanel : "St_ControlPanel";
   END_VAR
   VAR_OUTPUT
      LidClampClose : Bool;
      LidClampRise : Bool;
      BaseClampClose : Bool;
      BaseClampRise : Bool;
      AxisX : Bool;
      AxisZ : Bool;
      Grab : Bool;
   END_VAR
   VAR_IN_OUT
      "St_ Assembler" : "St_Assembler";
   END_VAR
   VAR
      iMachineState : Int;
      LidPresence : F_TRIG;
      BasePresence : F_TRIG;
      tVacuoOff : TON_TIME;
      tSaidaPeça : TON_TIME;
      tLidClampUp : TON_TIME;
      tLidClampDown : TON_TIME;
      tBaseClampUp : TON_TIME;
      tBaseClampDown : TON_TIME;
      tXFoward : TON_TIME;
      tXBackward : TON_TIME;
      tZRise : TON_TIME;
      tZDown : TON_TIME;
   END_VAR
BEGIN
   REGION Memory Presence
       #LidPresence(CLK := #PresenceLidConveyor); // PULSE LID PRESENCE
       IF #LidPresence.Q THEN
           #"St_ Assembler".MemoryPresenceLid := 1;
       END_IF;

       #BasePresence(CLK := #PresenceBaseConveyor); // PULSE BASE PRESENCE
       IF #BasePresence.Q THEN
           #"St_ Assembler".MemoryPresenceBase := 1;
       END_IF;
   END_REGION

   REGION HOME MACHINE
       IF #ControlPanel.q_xPanelResetCmd THEN
           #LidClampClose := 0;
           #LidClampRise := 0;
           #BaseClampClose := 0;
           #BaseClampRise := 0;
           #AxisX := 1;
           #AxisZ := 0;
           #Grab := 0;
           #"St_ Assembler".iMachineState := 0;
           #"St_ Assembler".MemoryPresenceLid := 0;
           #"St_ Assembler".MemoryPresenceBase := 0;
       END_IF;
   END_REGION

   REGION Timmers
       #tVacuoOff(IN := NOT #Grab,
                  PT := T#500ms);

       #tSaidaPeça(IN:=#BaseClampRise,
                   PT:=T#3s);

       #tLidClampUp(IN:=#LidClampRise AND #LidClampLimit ,
                    PT:=T#300ms,
                    Q=>#"St_ Assembler".LidClampUpPosition);

       #tLidClampDown(IN:=NOT #LidClampRise AND #LidClampLimit,
                      PT:=T#300ms,
                      Q=>#"St_ Assembler".LidClampDownPosition);

       #tBaseClampUp(IN:=#BaseClampRise AND #BaseClampLimit,
                     PT:=T#300ms,
                     Q=>#"St_ Assembler".BaseClampUpPosition);

       #tBaseClampDown(IN:=NOT #BaseClampRise AND #BaseClampLimit,
                       PT:=T#300ms,
                       Q=>#"St_ Assembler".BaseClampDownPosition);

       #tXFoward(IN:=#AxisX AND NOT #MovingX ,
                 PT:=T#300ms,
                 Q=>#"St_ Assembler".AxisXFoward);

       #tXBackward(IN:= NOT #AxisX AND NOT #MovingX,
                   PT:=T#300ms,
                   Q=>#"St_ Assembler".AxisXBackward);

       #tZRise(IN:=NOT #AxisZ AND NOT #MovingZ,
               PT:=T#300ms,
               Q=>#"St_ Assembler".AxisZRise);

       #tZDown(IN:=#AxisZ AND NOT #MovingZ,
               PT:=T#300ms,
               Q=>#"St_ Assembler".AxisZDown);
   END_REGION

   // READY TO RECEIVE SIGNAL
   #"St_ Assembler".ReadyToReceiveLid := #ControlPanel.q_xAutoMode AND #"St_ Assembler".iMachineState = 1 AND NOT #"St_ Assembler".MemoryPresenceLid;
   #"St_ Assembler".ReadyToReceiveBase := #ControlPanel.q_xAutoMode AND #"St_ Assembler".iMachineState = 1 AND NOT #"St_ Assembler".MemoryPresenceBase;
   IF #ControlPanel.q_xAutoMode THEN
       CASE #"St_ Assembler".iMachineState OF
           0:  // HOME MACHINE
               #"St_ Assembler".iState := 'S00 PASSO INICIAL';
               #LidClampClose := FALSE;
               #LidClampRise := FALSE;
               #BaseClampClose := FALSE;
               #BaseClampRise := FALSE;
               #AxisX := TRUE;
               #AxisZ := FALSE;
               #Grab := FALSE;

               IF NOT #LidClampClosed AND #"St_ Assembler".LidClampDownPosition AND NOT #BaseClampClosed AND #"St_ Assembler".BaseClampDownPosition AND #"St_ Assembler".AxisXFoward AND #"St_ Assembler".AxisZRise THEN
                   #"St_ Assembler".iMachineState := 1;
               END_IF;
               ;
           1:  // AGUARDANDO LID E BASE PRESENÇA
               #"St_ Assembler".iState := 'S01 AGUARDANDO LID E BASE PRESENCA';
               IF #"St_ Assembler".MemoryPresenceLid THEN
                   #LidClampClose := 1;
               END_IF;
               IF #"St_ Assembler".MemoryPresenceBase THEN
                   #BaseClampClose := 1;
               END_IF;
               IF #LidClampClosed AND #BaseClampClosed AND #"St_ Assembler".MemoryPresenceBase AND #"St_ Assembler".MemoryPresenceLid THEN
                   #"St_ Assembler".iMachineState := 2;
               END_IF;

           2: // PICK POSITION
               #"St_ Assembler".iState := 'S02 PICK POSITION';
               #AxisX := 1;
               IF #"St_ Assembler".AxisXFoward THEN
                   #AxisZ := 1;
               END_IF;
               IF #"St_ Assembler".AxisXFoward AND #"St_ Assembler".AxisZDown THEN
                   #"St_ Assembler".iMachineState := 3;
               END_IF;

           3: // ACIONA VACUO
               #"St_ Assembler".iState := 'S03 ACIONA VACUO';
               #Grab := 1;
               IF #Grab AND #PresenceGrab THEN
                   #"St_ Assembler".iMachineState := 4;
               END_IF;

           4: // RETIRA LID 
               #"St_ Assembler".iState := 'S04 RETIRA LID';
               #LidClampClose := 0;
               #AxisZ := 0;
               IF NOT #LidClampClosed AND #"St_ Assembler".AxisZRise AND #PresenceGrab THEN
                   #"St_ Assembler".MemoryPresenceLid := 0;
                   #"St_ Assembler".iMachineState := 5;
               END_IF;

           5: // RECUA EIXO X
               #"St_ Assembler".iState := 'S05 RECUA EIXO X';
               #AxisX := 0;
               IF #"St_ Assembler".AxisXBackward THEN
                   #"St_ Assembler".iMachineState := 6;
               END_IF;

           6: // DESCE PARA MONTAGEM
               #"St_ Assembler".iState := 'S06 DESCE PARA MONTAGEM';
               #AxisZ := 1;
               IF #"St_ Assembler".AxisZDown THEN
                   #"St_ Assembler".iMachineState := 7;
               END_IF;

           7: // LIBERA VACUO
               #"St_ Assembler".iState := 'S07 LIBERA VACUO';
               #Grab := 0;
               IF #tVacuoOff.Q THEN
                   #"St_ Assembler".iMachineState := 8;
               END_IF;

           8: // SOBE SEM PEÇA
               #"St_ Assembler".iState := 'S08 SOBE SEM PECA';
               #AxisZ := 0;
               #BaseClampClose := 0;
               IF NOT #BaseClampClosed AND #"St_ Assembler".AxisZRise AND NOT #PresenceGrab AND #"St_ Assembler".EnableSend THEN
                   #"St_ Assembler".iMachineState := 9;
               END_IF;

           9: // LIBERA PEÇA COMPLETA
               #"St_ Assembler".iState := 'S09 LIBERA PECA COMPLETA';
               #AxisX := 1;
               #BaseClampRise := 1;
               IF #"St_ Assembler".AxisXFoward AND #tSaidaPeça.Q THEN
                   #"St_ Assembler".MemoryPresenceBase := 0;
                   #"St_ Assembler".iMachineState := 0;
               END_IF;
           ELSE  
               #"St_ Assembler".iMachineState := 0; 
       END_CASE;
   END_IF;
END_FUNCTION_BLOCK

FUNCTION_BLOCK "Manipulator"   // FB14, SCL
{ S7_Optimized_Access := 'TRUE' }
VERSION : 0.1
   VAR_INPUT
      "Pallet Detected" : Bool;
      "Part Detected" : Bool;
      PresenceGrab : Bool;
      "Actual Position X" : Int;
      "Actual Position Y" : Int;
      "Actual Position Z" : Int;
      ControlPanel : "St_ControlPanel";
   END_VAR
   VAR_OUTPUT
      "X Setpoint" : Int;
      "Y Setpoint" : Int;
      "Z Setpoint" : Int;
      Grab : Bool;
   END_VAR
   VAR_IN_OUT
      Manipulator : "St_Manipulator";
   END_VAR
   VAR
      Position : Struct
         x : Int;
         y : Int;
         z : Int;
      END_STRUCT;
      "Null Position" : Bool;
      i : Int;
      GrabOff : TON_TIME;
      NotPallet : TON_TIME;
   END_VAR
   VAR CONSTANT
      Tolerance : Int := 30;
      Offset : Int := -2000;
   END_VAR
   // // Manipulator.Coordinates[0] : Home
   // // Manipulator.Coordinates[1] : PrePick
   // // Manipulator.Coordinates[2] : Pick
   // // Manipulator.Coordinates[3] : PosPick
   // // Manipulator.Coordinates[4] : PreDrop
   // // Manipulator.Coordinates[5] : Drop
   // // Manipulator.Coordinates[6] : PosDrop
   // // Manipulator.Ack_Positions[0] : Home
   // // Manipulator.Ack_Positions[1] : PrePick
   // // Manipulator.Ack_Positions[2] : Pick
   // // Manipulator.Ack_Positions[3] : PosPick
   // // Manipulator.Ack_Positions[4] : PreDrop
   // // Manipulator.Ack_Positions[5] : Drop
   // // Manipulator.Ack_Positions[6] : PosDrop
BEGIN

   REGION "General" Reset
       IF #ControlPanel.q_xPanelResetCmd THEN
           #Position := #Manipulator.Coordinates[0]; //Home
           #Grab := 0;
           #Manipulator.ReadyToReceivePallet := 0;
           #Manipulator.PalletFull := 0;
           #Manipulator.ContActual := 0;
           #Manipulator.iMachineState := 0;
       END_IF;

   END_REGION

   REGION Timers
       #GrabOff(IN:=NOT #Grab, PT:=T#1s);
       #NotPallet(IN:=NOT #"Pallet Detected", PT:=T#2s);
   END_REGION

   REGION Acknowledged Position      
       // "General".Manipulator.Coordinates[5]."Axis Z" := 27648 - (#Manipulator.ContActual * 2000);
       FOR #i := 0 TO "MaxCoordinates" DO
           #Manipulator.Ack_Positions[#i] := "Ack Position"("Actual Position X" := #"Actual Position X",
                                                            "Actual Position Y" := #"Actual Position Y",
                                                            "Actual Position Z" := #"Actual Position Z",
                                                            Position := #Manipulator.Coordinates[#i]);
       END_FOR;
   END_REGION

   REGION Machine State
       IF #ControlPanel.q_xAutoMode THEN

           CASE #Manipulator.iMachineState OF
               0:  // RESET CONTADOR
                   #Manipulator.iState := 'S00 PASSO INICIAL';
                   #Manipulator.ContActual := 0;
                   #Manipulator.ReadyToReceivePallet := 0;
                   #Manipulator.PalletFull := 0;
                   IF #Manipulator.ContActual = 0 THEN
                       #Manipulator.iMachineState := 1;
                   END_IF;

               1: // HOME MACHINE 
                   #Manipulator.iState := 'S01 POSICAO INICIAL';
                       #Position := #Manipulator.Coordinates[0];
                       #Grab := 0;
                       IF #Manipulator.Ack_Positions[0] AND NOT #PresenceGrab THEN
                       #Manipulator.iMachineState := 2;
                   END_IF;

               2: // AGUARDANDO PALET E PEÇA
                   #Manipulator.iState := 'S02 AGUARDANDO PALET E PEÇA';
                   #Manipulator.ReadyToReceivePallet := 1;

                   IF #"Pallet Detected" THEN
                       #Manipulator.ReadyToReceivePallet := 0;    
                   END_IF;

                   IF #"Pallet Detected" AND #"Part Detected" THEN
                       #Manipulator.iMachineState := 3;
                       #Manipulator.ReadyToReceivePallet := 0;
                   END_IF;

               3: // PREPICK POSITION
                   #Manipulator.iState := 'S03 PREPICK POSITION';
                   #Position := #Manipulator.Coordinates[1];
                   IF #Manipulator.Ack_Positions[1] THEN
                       #Manipulator.iMachineState := 4;
                   END_IF;

               4: // PICK POSITION
                   #Manipulator.iState := 'S04 PICK POSITION';
                   #Position := #Manipulator.Coordinates[2];
                   IF #Manipulator.Ack_Positions[2] THEN
                       #Manipulator.iMachineState := 5;
                   END_IF;

               5: // LIGAR VACUO 
                   #Manipulator.iState := 'S05 LIGAR VACUO';
                   #Grab := 1;
                   IF #Grab AND #PresenceGrab THEN
                       #Manipulator.iMachineState := 6;
                   END_IF;

               6: // POSPICK POSITION
                   #Manipulator.iState := 'S06 POSPICK POSITION';
                   #Position := #Manipulator.Coordinates[3];
                   IF #Manipulator.Ack_Positions[3] AND #PresenceGrab THEN
                       #Manipulator.iMachineState := 7;
                   END_IF;

               7: //PREDROP POSITION
                   #Manipulator.iState := 'S07 PREDROP POSITION';
                   #Position := #Manipulator.Coordinates[4];
                   IF #Manipulator.Ack_Positions[4] AND #"Pallet Detected" THEN
                       #Manipulator.iMachineState := 8;
                   END_IF;

               8: //DROP POSITION
                   #Manipulator.iState := 'S08 DROP POSITION';
                   #Position := #Manipulator.Coordinates[5];
                   IF #Manipulator.Ack_Positions[5] THEN
                       #Manipulator.iMachineState := 9;
                   END_IF;

               9: // LIBERA VACUO
                   #Manipulator.iState := 'S09 LIBERA VACUO';
                   #Grab := 0;
                   IF #GrabOff.Q THEN
                       #Manipulator.iMachineState := 10;
                   END_IF;

               10: // POS DROP
                   #Manipulator.iState := 'S10 POS DROP';
                   #Position := #Manipulator.Coordinates[6];
                   IF #Manipulator.Ack_Positions[6] AND NOT #PresenceGrab THEN
                       #Manipulator.ContActual := #Manipulator.ContActual + 1;
                       #Manipulator.iMachineState := 11;
                   END_IF;

               11: // VERIFICA CONTADOR
                   #Manipulator.iState := 'S11 VERIFICA CONTADOR';
                   IF #Manipulator.ContActual >= #Manipulator.ContMax THEN

                       #Manipulator.iMachineState := 12;
                   ELSE
                       #Manipulator.iMachineState := 1;
                   END_IF;

               12: //PALET CHEIO
                   #Manipulator.iState := 'S12 PALET CHEIO';
                   #Manipulator.PalletFull := 1;
                   IF #NotPallet.Q THEN
                       #Manipulator.iMachineState := 0;
                   END_IF;
               ELSE  
                   #Manipulator.iMachineState := 0;
           END_CASE;
       END_IF;
   END_REGION

   REGION OFFSET FROP


   END_REGION


   REGION OUTPUTS
       #"X Setpoint" := #Position.x;
       #"Y Setpoint" := #Position.y;
       #"Z Setpoint" := #Position.z;
   END_REGION
END_FUNCTION_BLOCK

FUNCTION_BLOCK "Transfer"   // FB15, SCL
{ S7_Optimized_Access := 'TRUE' }
VERSION : 0.1
   VAR_INPUT
      RightStop : Bool;
      LeftStop : Bool;
      ControlPanel : "St_ControlPanel";
   END_VAR
   VAR_OUTPUT
      "Chain Transfer Foward" : Bool;
      "Chain Transfer Backward" : Bool;
      "Chain Transfer Right" : Bool;
      "Chain Transfer Left" : Bool;
   END_VAR
   VAR_IN_OUT
      Transfer : "St_Transfer";
   END_VAR
BEGIN

   REGION Reset    
       IF #ControlPanel.q_xPanelResetCmd THEN
           #Transfer.iMachineState := 0;
           #Transfer."Chain Transfer Foward" := 0;
           #Transfer."Chain Transfer Backward" := 0;
           #Transfer."Chain Transfer Right" := 0;
           #Transfer."Chain Transfer Left" := 0;
           #Transfer.ReadyToReceiveRight := 0;
           #Transfer.ReadyToReceiveLeft := 0;
       END_IF;
   END_REGION


   REGION Machine State    
       IF #ControlPanel.q_xAutoMode THEN
           CASE #Transfer.iMachineState OF
               0:  // HOME 
                   #Transfer.iState := 'S00 HOME POSITION';
                   #Transfer."Chain Transfer Foward" := 0;
                   #Transfer."Chain Transfer Backward" := 0;
                   #Transfer."Chain Transfer Right" := 0;
                   #Transfer."Chain Transfer Left" := 0;
                   #Transfer.ReadyToReceiveRight := 0;
                   #Transfer.ReadyToReceiveLeft := 0;

                   IF NOT #RightStop AND NOT #LeftStop THEN
                       #Transfer.iMachineState := 1;
                   END_IF;

               1:  // AGUARDA PALET
                   #Transfer.iState := 'S01 AGUARDA PALET';

                   IF #Transfer.RequestRight AND NOT #Transfer.RequestLeft THEN
                       #Transfer.iMachineState := 2;
                   ELSIF NOT #Transfer.RequestRight AND #Transfer.RequestLeft THEN
                       #Transfer.iMachineState := 3;
                   ELSIF #Transfer.RequestRight AND #Transfer.RequestLeft THEN
                       IF #Transfer.LastReceiveRightSide THEN
                           #Transfer.iMachineState := 3;
                       ELSE
                           #Transfer.iMachineState := 2;
                       END_IF;
                   END_IF;

               2: // RECEBE PALET PELA DIREITA
                   #Transfer.iState := 'S02 RECEBE PALET PELA DIREITA';
                   #Transfer.ReadyToReceiveRight := 1;
                   #Transfer."Chain Transfer Right" := 1;
                   IF #RightStop THEN
                       #Transfer.iMachineState := 4;
                       #Transfer.LastReceiveRightSide := 1;
                   END_IF;

               3: // RECEBE PALET PELA ESQUERDA
                   #Transfer.iState := 'S03 RECEBE PALET PELA ESQUERDA';
                   #Transfer.ReadyToReceiveLeft := 1;
                   #Transfer."Chain Transfer Left" := 1;
                   IF #LeftStop THEN
                       #Transfer.iMachineState := 4;
                       #Transfer.LastReceiveRightSide := 0;
                   END_IF;

               4: // AGUARDA LIBERACAO PARA ENVIAR
                   #Transfer.iState := 'S04 AGUARDA LIBERACAO PARA ENVIAR';
                   #Transfer.ReadyToReceiveLeft := 0;
                   #Transfer.ReadyToReceiveRight := 0;
                   #Transfer."Chain Transfer Right" := 0;
                   #Transfer."Chain Transfer Left" := 0;
                   IF #Transfer.EnableSend THEN
                       #Transfer.iMachineState := 5;
                   END_IF;

               5: // ENVIAR PALET 
                   #Transfer.iState := 'S05 AGUARDA LIBERACAO PARA ENVIAR';
                   #Transfer."Chain Transfer Foward" := 1;
                   IF NOT #Transfer.EnableSend THEN
                       #Transfer.iMachineState := 0;
                   END_IF;

               ELSE
                   #Transfer.iMachineState := 0;
           END_CASE;
       END_IF;
   END_REGION

   REGION OUTPUTS
       CASE #ControlPanel.q_siMode OF
           1:  // EMERGENCIA
               #"Chain Transfer Foward" := 0;
               #"Chain Transfer Backward" := 0;
               #"Chain Transfer Right" := 0;
               #"Chain Transfer Left" := 0;

           2:  // AUTOMATICO
               #"Chain Transfer Foward" := #Transfer."Chain Transfer Foward";
               #"Chain Transfer Backward" := #Transfer."Chain Transfer Backward";
               #"Chain Transfer Right" := #Transfer."Chain Transfer Right";
               #"Chain Transfer Left" := #Transfer."Chain Transfer Left";

           3:  // MANUAL
               #"Chain Transfer Foward" := 0;
               #"Chain Transfer Backward" := 0;
               #"Chain Transfer Right" := 0;
               #"Chain Transfer Left" := 0;

           ELSE
               #"Chain Transfer Foward" := 0;
               #"Chain Transfer Backward" := 0;
               #"Chain Transfer Right" := 0;
               #"Chain Transfer Left" := 0;
       END_CASE;
   END_REGION
END_FUNCTION_BLOCK

FUNCTION "PosDisponivel" : DInt   // FC1, SCL
{ S7_Optimized_Access := 'TRUE' }
VERSION : 0.1
   VAR_INPUT
      Armazem : Array[1..54] of Bool;
   END_VAR
   VAR_TEMP
      i : Int;
      j : Int;
      "Array" : Array[1..54] of Int;
   END_VAR
   VAR CONSTANT
      Inicio : Int := 1;
      Fim : Int := 54;
   END_VAR
BEGIN
   //INICIALIZA VARIAVEL
   #PosDisponivel := -1;

   //PRIORIDADE ABASTECIMENTO
   #Array[1] := 1;
   #Array[2] := 10;
   #Array[3] := 19;
   #Array[4] := 28;
   #Array[5] := 37;
   #Array[6] := 46;

   #Array[7] := 2;
   #Array[8] := 11;
   #Array[9] := 20;
   #Array[10] := 29;
   #Array[11] := 38;
   #Array[12] := 47;

   #Array[13] := 3;
   #Array[14] := 12;
   #Array[15] := 21;
   #Array[16] := 30;
   #Array[17] := 39;
   #Array[18] := 48;

   #Array[19] := 4;
   #Array[20] := 13;
   #Array[21] := 22;
   #Array[22] := 31;
   #Array[23] := 40;
   #Array[24] := 49;

   #Array[25] := 5;
   #Array[26] := 14;
   #Array[27] := 23;
   #Array[28] := 32;
   #Array[29] := 41;
   #Array[30] := 50;

   #Array[31] := 6;
   #Array[32] := 15;
   #Array[33] := 24;
   #Array[34] := 33;
   #Array[35] := 42;
   #Array[36] := 51;

   #Array[37] := 7;
   #Array[38] := 16;
   #Array[39] := 25;
   #Array[40] := 34;
   #Array[41] := 43;
   #Array[42] := 52;

   #Array[43] := 8;
   #Array[44] := 17;
   #Array[45] := 26;
   #Array[46] := 35;
   #Array[47] := 44;
   #Array[48] := 53;

   #Array[49] := 9;
   #Array[50] := 18;
   #Array[51] := 27;
   #Array[52] := 36;
   #Array[53] := 45;
   #Array[54] := 54;

   //PROCURA POSICAO LIVRE
   FOR #i := #Inicio TO #Fim DO
       #j := #Array[#i];
       IF NOT #Armazem[#j] THEN
           #PosDisponivel := INT_TO_DINT(#j);
           EXIT;
       END_IF;
   END_FOR;
END_FUNCTION

FUNCTION "Ack Position" : Bool   // FC2, SCL
{ S7_Optimized_Access := 'TRUE' }
VERSION : 0.1
   VAR_INPUT
      "Actual Position X" : Int;
      "Actual Position Y" : Int;
      "Actual Position Z" : Int;
      Position : Struct
         x : Int;
         y : Int;
         z : Int;
      END_STRUCT;
   END_VAR
   VAR_TEMP
      Null : Bool;
   END_VAR
   VAR CONSTANT
      Tolerance : Int := 30;
   END_VAR
BEGIN

   #Null := #"Actual Position X" = 0 OR #"Actual Position Y" = 0 OR #"Actual Position Z" = 0;

   #"Ack Position" := NOT #Null

   AND #"Actual Position X" >= #Position.x - #Tolerance AND #"Actual Position X" <= #Position.x + #Tolerance
   AND #"Actual Position Y" >= #Position.y - #Tolerance AND #"Actual Position Y" <= #Position.y + #Tolerance
   AND #"Actual Position Z" >= #Position.z - #Tolerance AND #"Actual Position Z" <= #Position.z + #Tolerance;
END_FUNCTION

FUNCTION "MHJ-PLC-Lab-Function-S71200" : Void   // FC9000, SCL
{ S7_Optimized_Access := 'TRUE' }
VERSION : 0.1
   VAR_TEMP
      rdTimeReturn : Int;
      outputTime : DTL;
      SyncVal : Byte;
      forVal : Int;
      forVal_2 : Int;
      Value : Byte;
   END_VAR
   VAR CONSTANT
      CompVal : Byte := 16#34;
      Value_01 : Byte := 16#11;
      Value_01_DW : DWord := 16#A165_D992;
      Value_02_DW : DWord := 16#58BE_4401;
   END_VAR
BEGIN

   #Value:=PEEK(area := 16#82,
        dbNumber := 0,
        byteOffset := 511);
   #Value := #Value + 1;

   POKE(area := 16#82,
        dbNumber := 0,
        byteOffset := 511,
        value := #Value);

   POKE(area:=16#81,
        dbNumber:=0,
        byteOffset:=1016,
        value:=#Value_01_DW);
   POKE(area := 16#81,
        dbNumber := 0,
        byteOffset := 1020,
        value := #Value_02_DW);

   POKE(area := 16#81,
        dbNumber := 0,
        byteOffset := 511,
        value := B#16#00);

   FOR #forVal := 0 TO 120 DO
       FOR #forVal_2:=0 TO 10 DO
           #rdTimeReturn:=RD_SYS_T(#outputTime);
           #rdTimeReturn := WR_SYS_T(#outputTime);
           #rdTimeReturn := RD_SYS_T(#outputTime);
           #rdTimeReturn := WR_SYS_T(#outputTime);
       END_FOR;
       #SyncVal:= PEEK(area := 16#81,
                      dbNumber := 0,
                      byteOffset := 511);
       IF #SyncVal = #CompVal THEN
          GOTO M_1;
       END_IF;
   END_FOR;
   RETURN;

   M_1:
   POKE(area := 16#81,
        dbNumber := 0,
        byteOffset := 511,
        value := B#16#0);
END_FUNCTION

// folder: ZNE01

FUNCTION_BLOCK "Zne01"   // FB4, SCL
{ S7_Optimized_Access := 'TRUE' }
VERSION : 0.1
   VAR
      "Sorter 102" : "Sorter";
      "Sorter 123" : "Sorter";
      "Conveyor 101" : "Conveyor";
      "Conveyor 120" : "Conveyor";
      "Conveyor 121" : "Conveyor";
      "Conveyor 122" : "Conveyor";
      "Conveyor 124" : "Conveyor";
      "Conveyor 125" : "Conveyor";
      Aux_xLastPartCenter0 : Bool;
      Aux_xLastPartCenter2 : Bool;
      "Machine Center 0" : "MachineCenter";
      "Machine Center 1" : "MachineCenter";
      "Conveyor 130" : "Conveyor";
      "Conveyor 131" : "Conveyor";
      "Conveyor 132" : "Conveyor";
      "Sorter 133" : "Sorter";
      "Conveyor 134" : "Conveyor";
      "Conveyor 135" : "Conveyor";
      "Machine Center 2" : "MachineCenter";
      "Machine Center 3" : "MachineCenter";
      tInterlockConveyor122 : TOF_TIME;
      tInterlockConveyor132 : TOF_TIME;
   END_VAR
BEGIN


   REGION #"Conveyor 101"
       #"Conveyor 101".i_xInterlock := (#"Sorter 102".i_xRightRequest AND NOT #"Conveyor 120".q_xMotorOn) OR (#"Sorter 102".i_xLeftRequest AND NOT #"Conveyor 130".q_xMotorOn);
       #"Conveyor 101"(i_xRun := TRUE,
                       ControlPanel := "General".Panel01,
                       q_xMotorOn => "Zne01 Conveyor 101",
                       Conveyor := "General"."Conveyor 101");
   END_REGION

   REGION #"Sorter 102"
       #"Sorter 102".i_xRightRequest := "Vision Sensor 0 (Value)" = "GreenRawMaterial";
       #"Sorter 102".i_xLeftRequest := "Vision Sensor 0 (Value)" = "BlueRawMaterial";
       #"Sorter 102".i_xCenterRequest := ("Vision Sensor 0 (Value)" <> "BlueRawMaterial") AND ("Vision Sensor 0 (Value)" <> "GreenRawMaterial") AND ("Vision Sensor 0 (Value)" <> 0);
       #"Sorter 102"(ControlPanel := "General".Panel01,
                     q_xUp => "Zne01 Sorter 102 (Up)",
                     q_xRight => "Zne01 Sorter 102 (Right)",
                     q_xLeft => "Zne01 Sorter 102 (Left)");
   END_REGION

   REGION #"Conveyor 120"
       #"Conveyor 120".i_xInterlock := "Sensor 120" AND NOT #"Conveyor 121".q_xMotorOn;
       #"Conveyor 120"(i_xRun := TRUE,
                       ControlPanel := "General".Panel01,
                       q_xMotorOn => "Zne01 Conveyor 120",
                       Conveyor := "General"."Conveyor 120");
   END_REGION

   REGION #"Conveyor 121"    
       #"Conveyor 121".i_xInterlock := NOT #"Conveyor 122".q_xMotorOn;
       #"Conveyor 121"(i_xRun := TRUE,
                       ControlPanel := "General".Panel01,
                       q_xMotorOn => "Zne01 Conveyor 121",
                       Conveyor := "General"."Conveyor 121");
   END_REGION

   REGION #"Conveyor 122"
       #tInterlockConveyor122(IN:="Sensor 122" AND ((NOT #"Conveyor 124".q_xMotorOn AND "Zne01 Sorter 123 (Right)") OR (NOT #"Conveyor 125".q_xMotorOn AND NOT "Zne01 Sorter 123 (Right)")),
                              PT:=T#2s);

       #"Conveyor 122".i_xInterlock := #tInterlockConveyor122.Q;
       #"Conveyor 122"(i_xRun := TRUE,
                       ControlPanel := "General".Panel01,
                       q_xMotorOn => "Zne01 Conveyor 122",
                       Conveyor := "General"."Conveyor 122");
   END_REGION

   REGION #"Sorter 123"

       //DIRECTION LOGIC
       IF NOT "Machining Center 0 (Is Busy)" AND "Machining Center 1 (Is Busy)" THEN
           #"Sorter 123".i_xRightRequest := TRUE;
           #"Sorter 123".i_xCenterRequest := FALSE;
       ELSIF "Machining Center 0 (Is Busy)" AND NOT "Machining Center 1 (Is Busy)" THEN
           #"Sorter 123".i_xRightRequest := FALSE;
           #"Sorter 123".i_xCenterRequest := TRUE;
       ELSIF NOT "Machining Center 0 (Is Busy)" AND NOT "Machining Center 1 (Is Busy)" THEN
           IF #Aux_xLastPartCenter0 THEN
               #"Sorter 123".i_xRightRequest := FALSE;
               #"Sorter 123".i_xCenterRequest := TRUE;
           ELSE
               #"Sorter 123".i_xRightRequest := TRUE;
               #"Sorter 123".i_xCenterRequest := FALSE;
           END_IF;
       END_IF;

       //LAST PART MEMORY DIRECTION
       IF "Machining Center 0 (Is Busy)" THEN
           #Aux_xLastPartCenter0 := TRUE;
       ELSIF "Machining Center 1 (Is Busy)" THEN
           #Aux_xLastPartCenter0 := FALSE;
       END_IF;

       #"Sorter 123"(ControlPanel := "General".Panel01,
                     q_xUp => "Zne01 Sorter 123 (Up)",
                     q_xRight => "Zne01 Sorter 123 (Right)");
   END_REGION

   REGION #"Conveyor 124"
       #"Conveyor 124".i_xInterlock := "Machining Center 0 (Is Busy)";
       #"Conveyor 124"(i_xRun := TRUE,
                       ControlPanel := "General".Panel01,
                       q_xMotorOn => "Zne01 Conveyor 124",
                       Conveyor := "General"."Conveyor 124");
   END_REGION

   REGION #"Conveyor 125"    
       #"Conveyor 125".i_xInterlock := "Machining Center 1 (Is Busy)" OR #"Machine Center 1".Interlock;
       #"Conveyor 125"(i_xRun := TRUE,
                       ControlPanel := "General".Panel01,
                       q_xMotorOn => "Zne01 Conveyor 125",
                       Conveyor := "General"."Conveyor 125");
   END_REGION

   REGION #"Machine Center 0"    
       #"Machine Center 0"(Interlock := FALSE,
                           ControlPanel := "General".Panel01,
                           Start => "Machining Center 0 (Start)",
                           Stop => "Machining Center 0 (Stop)",
                           Reset => "Machining Center 0 (Reset)");
   END_REGION

   REGION #"Machine Center 1"
       #"Machine Center 1"(Interlock := NOT "Zne03 Conveyor 300",
                           ControlPanel := "General".Panel01,
                           Start => "Machining Center 1 (Start)",
                           Stop => "Machining Center 1 (Stop)",
                           Reset => "Machining Center 1 (Reset)");
   END_REGION

   REGION #"Conveyor 130"
       #"Conveyor 130".i_xInterlock := "Sensor 130" AND NOT #"Conveyor 131".q_xMotorOn;
       #"Conveyor 130"(i_xRun := TRUE,
                       ControlPanel := "General".Panel01,
                       q_xMotorOn => "Zne01 Conveyor 130",
                       "Conveyor" := "General"."Conveyor 130");
   END_REGION

   REGION #"Conveyor 131"
       #"Conveyor 131".i_xInterlock := NOT #"Conveyor 132".q_xMotorOn;
       #"Conveyor 131"(i_xRun := TRUE,
                       ControlPanel := "General".Panel01,
                       q_xMotorOn => "Zne01 Conveyor 131",
                       Conveyor := "General"."Conveyor 131");
   END_REGION

   REGION #"Conveyor 132"    
       #tInterlockConveyor132(IN := "Sensor 132" AND ((NOT #"Conveyor 134".q_xMotorOn AND "Zne01 Sorter 133 (Left)") OR (NOT #"Conveyor 135".q_xMotorOn AND NOT "Zne01 Sorter 133 (Left)")),
                              PT := T#2s);
       #"Conveyor 132".i_xInterlock := #tInterlockConveyor132.Q;
       #"Conveyor 132"(i_xRun := TRUE,
                       ControlPanel := "General".Panel01,
                       q_xMotorOn => "Zne01 Conveyor 132",
                       Conveyor := "General"."Conveyor 132");
   END_REGION

   REGION #"Sorter 133"

       //DIRECTION LOGIC
       IF NOT "Machining Center 2 (Is Busy)" AND "Machining Center 3 (Is Busy)" THEN
           #"Sorter 133".i_xCenterRequest := TRUE;
           #"Sorter 133".i_xLeftRequest := FALSE;
       ELSIF "Machining Center 2 (Is Busy)" AND NOT "Machining Center 3 (Is Busy)" THEN
           #"Sorter 133".i_xCenterRequest := FALSE;
           #"Sorter 133".i_xLeftRequest := TRUE;
       ELSIF NOT "Machining Center 2 (Is Busy)" AND NOT "Machining Center 3 (Is Busy)" THEN
           IF #Aux_xLastPartCenter2 THEN
               #"Sorter 133".i_xCenterRequest := FALSE;
               #"Sorter 133".i_xLeftRequest := TRUE;
           ELSE
               #"Sorter 133".i_xCenterRequest := TRUE;
               #"Sorter 133".i_xLeftRequest := FALSE;
           END_IF;
       END_IF;

       //LAST PART MEMORY DIRECTION
       IF "Machining Center 2 (Is Busy)" THEN
           #Aux_xLastPartCenter2 := TRUE;
       ELSIF "Machining Center 3 (Is Busy)" THEN
           #Aux_xLastPartCenter2 := FALSE;
       END_IF;

       #"Sorter 133"(ControlPanel := "General".Panel01,
                     q_xUp => "Zne01 Sorter 133 (Up)",
                     q_xLeft => "Zne01 Sorter 133 (Left)");
   END_REGION

   REGION #"Conveyor 134"
       #"Conveyor 134".i_xInterlock := "Machining Center 3 (Is Busy)";
       #"Conveyor 134"(i_xRun := TRUE,
                       ControlPanel := "General".Panel01,
                       q_xMotorOn => "Zne01 Conveyor 134",
                       Conveyor := "General"."Conveyor 134");
   END_REGION

   REGION #"Conveyor 135"
       #"Conveyor 135".i_xInterlock := "Machining Center 2 (Is Busy)" OR #"Machine Center 2".Interlock;
       #"Conveyor 135"(i_xRun := TRUE,
                       ControlPanel := "General".Panel01,
                       q_xMotorOn => "Zne01 Conveyor 135",
                       Conveyor := "General"."Conveyor 135");
   END_REGION

   REGION #"Machine Center 2"
       #"Machine Center 2"(Interlock := NOT "Zne05 Conveyor 500",
                           ControlPanel := "General".Panel01,
                           Start => "Machining Center 2 (Start)",
                           Stop => "Machining Center 2 (Stop)",
                           Reset => "Machining Center 2 (Reset)");
   END_REGION

   REGION #"Machine Center 3"
       #"Machine Center 3"(Interlock := FALSE,
                           ControlPanel := "General".Panel01,
                           Start => "Machining Center 3 (Start)",
                           Stop => "Machining Center 3 (Stop)",
                           Reset => "Machining Center 3 (Reset)");
   END_REGION
END_FUNCTION_BLOCK

// folder: ZNE02

FUNCTION_BLOCK "Zne02"   // FB7, SCL
{ S7_Optimized_Access := 'TRUE' }
VERSION : 0.1
   VAR
      "Conveyor 220" : "Conveyor";
      "Conveyor 221" : "Conveyor";
      "Pusher Zne02" : "Pusher";
      "Conveyor 222" : "Conveyor";
      "Conveyor 223" : "Conveyor";
      "Conveyor 224" : "Conveyor";
      "Conveyor 225" : "Conveyor";
   END_VAR
BEGIN

   REGION #"Conveyor 220"
       #"Conveyor 220"(i_xRun := TRUE,
                       ControlPanel := "General".Panel01,
                       q_xMotorOn => "Zne02 Conveyor 220",
                       Conveyor := "General"."Conveyor 220");
   END_REGION

   REGION #"Conveyor 221"
       #"Conveyor 221"(i_xRun:=TRUE,
                       ControlPanel:="General".Panel01,
                       q_xMotorOn=>"Zne02 Conveyor 221",
                       Conveyor:="General"."Conveyor 221");
   END_REGION

   REGION #"Pusher Zne02"    
       #"Pusher Zne02".RequestPusher := ("Vision Sensor 2 (Value)" <> "GreenLidMaterial") AND ("Vision Sensor 2 (Value)" <> 0);
       #"Pusher Zne02"(Timer := T#500ms,
                       "ControlPanel" := "General".Panel01,
                       Pusher => "Zne02 Pusher");
   END_REGION

   REGION #"Conveyor 222"    
       #"Conveyor 222"(i_xRun:=TRUE,
                       ControlPanel:="General".Panel01,
                       Conveyor:="General"."Conveyor 222");
       "Zne02 Conveyor 222A" := #"Conveyor 222".q_xMotorOn;
       "Zne02 Conveyor 222B" := #"Conveyor 222".q_xMotorOn;
   END_REGION

   REGION #"Conveyor 223"
       #"Conveyor 223".i_xInterlock := "Sensor 223" AND NOT "General"."Assembler Zne03".ReadyToReceiveLid;
       #"Conveyor 223"(i_xRun:=TRUE,
                       ControlPanel:="General".Panel01,
                       q_xMotorOn=>"Zne02 Conveyor 223",
                       Conveyor:="General"."Conveyor 223");
   END_REGION

   REGION #"Conveyor 224"
       #"Conveyor 224".i_xInterlock := FALSE;
       #"Conveyor 224"(i_xRun:=TRUE,
                       ControlPanel:="General".Panel01,
                       q_xMotorOn=>"Zne02 Conveyor 224",
                       Conveyor:="General"."Conveyor 224");
   END_REGION

   REGION "Conveyor 225"    
       #"Conveyor 225".i_xInterlock := FALSE;
   #"Conveyor 225"(i_xRun:=TRUE,
                   ControlPanel:="General".Panel01,
                   q_xMotorOn=>"Zne02 Conveyor 225",
                   Conveyor:="General"."Conveyor 225");
   END_REGION
END_FUNCTION_BLOCK

// folder: ZNE03

FUNCTION_BLOCK "Zne03"   // FB9, SCL
{ S7_Optimized_Access := 'TRUE' }
VERSION : 0.1
   VAR
      "Conveyor 300" : "Conveyor";
      "Conveyor 301" : "Conveyor";
      "Conveyor 302" : "Conveyor";
      "Pusher Zne03" : "Pusher";
      "Assembler Zne03" : "Assembler";
   END_VAR
BEGIN

   REGION "Conveyor 300"
       #"Conveyor 300".i_xInterlock := (NOT "General"."Assembler Zne03".ReadyToReceiveBase) AND "Sensor 300";
       #"Conveyor 300"(i_xRun:=TRUE,
                       ControlPanel:="General".Panel01,
                       q_xMotorOn=>"Zne03 Conveyor 300",
                       Conveyor:="General"."Conveyor 300");
   END_REGION

   REGION "Conveyor 301"
       #"Conveyor 301".i_xInterlock := FALSE;
       #"Conveyor 301"(i_xRun := TRUE,
                       ControlPanel := "General".Panel01,
                       q_xMotorOn => "Zne03 Conveyor 301",
                       Conveyor := "General"."Conveyor 301");
   END_REGION

   REGION "Conveyor 302"
       #"Conveyor 302".i_xInterlock := FALSE;
       #"Conveyor 302"(i_xRun := TRUE,
                       ControlPanel := "General".Panel01,
                       q_xMotorOn => "Zne03 Conveyor 302",
                       Conveyor := "General"."Conveyor 302");
   END_REGION

   REGION "Pusher Zne03"
       #"Pusher Zne03".RequestPusher := ("Vision Sensor 1 (Value)" <> "GreenBaseMaterial") AND ("Vision Sensor 1 (Value)" <> 0);
       #"Pusher Zne03"(Timer := T#500ms,
                       ControlPanel := "General".Panel01,
                       Pusher => "Zne03 Pusher");
   END_REGION

   REGION "Assembler"     
       "General"."Assembler Zne03".EnableSend := #"Conveyor 302".q_xMotorOn AND NOT "Sensor 302";
       #"Assembler Zne03"(LidClampClosed:="Zne02 Clamp Closed",
                          LidClampLimit:="Zne02 Clamp Limit",
                          BaseClampClosed:="Zne03 Clamp Closed",
                          BaseClampLimit:="Zne03 Clamp Limit",
                          PresenceLidConveyor:="Sensor 225",
                          PresenceBaseConveyor:="Sensor 301",
                          PresenceGrab:="Zne03 (Detected)",
                          MovingX:="Zne03 (Moving X)",
                          MovingZ:="Zne03 (Moving Z)",
                          ControlPanel:="General".Panel01,
                          LidClampClose=>"Zne02 Clamp",
                          LidClampRise=>"Zne02 Clamp Rise",
                          BaseClampClose=>"Zne03 Clamp",
                          BaseClampRise=>"Zne03 Clamp Raise",
                          AxisX=>"Zne03 X",
                          AxisZ=>"Zne03 Z",
                          Grab=>"Zne03 (Grab)",
                          "St_ Assembler":="General"."Assembler Zne03");
   END_REGION
END_FUNCTION_BLOCK

// folder: ZNE04

FUNCTION_BLOCK "Zne04"   // FB11, SCL
{ S7_Optimized_Access := 'TRUE' }
VERSION : 0.1
   VAR
      "Conveyor 420" : "Conveyor";
      "Conveyor 421" : "Conveyor";
      "Pusher Zne04" : "Pusher";
      "Conveyor 422" : "Conveyor";
      "Conveyor 423" : "Conveyor";
      "Conveyor 424" : "Conveyor";
      "Conveyor 425" : "Conveyor";
   END_VAR
BEGIN

   REGION "Conveyor 420"
       #"Conveyor 420"(i_xRun := TRUE,
                       ControlPanel := "General".Panel01,
                       q_xMotorOn => "Zne04 Conveyor 420",
                       Conveyor := "General"."Conveyor 420");
   END_REGION

   REGION "Conveyor 421"
       #"Conveyor 421"(i_xRun := TRUE,
                       ControlPanel := "General".Panel01,
                       q_xMotorOn => "Zne04 Conveyor 421",
                       Conveyor := "General"."Conveyor 421");
   END_REGION

   REGION 4"Pusher Zne04"    
       #"Pusher Zne04".RequestPusher := ("Vision Sensor 4 (Value)" <> "BlueLidMaterial") AND ("Vision Sensor 4 (Value)" <> 0);
       #"Pusher Zne04"(Timer := T#500ms,
                       "ControlPanel" := "General".Panel01,
                       Pusher => "Zne04 Pusher");
   END_REGION

   REGION "Conveyor 422"    
       #"Conveyor 422"(i_xRun := TRUE,
                       ControlPanel := "General".Panel01,
                       Conveyor := "General"."Conveyor 422");
       "Zne04 Conveyor 422A" := #"Conveyor 422".q_xMotorOn;
       "Zne04 Conveyor 422B" := #"Conveyor 422".q_xMotorOn;
   END_REGION

   REGION "Conveyor 423"
       #"Conveyor 423".i_xInterlock := "Sensor 423" AND NOT "General"."Assembler Zne05".ReadyToReceiveLid;
       #"Conveyor 423"(i_xRun := TRUE,
                       ControlPanel := "General".Panel01,
                       q_xMotorOn => "Zne04 Conveyor 423",
                       Conveyor := "General"."Conveyor 423");
   END_REGION

   REGION "Conveyor 424"
       #"Conveyor 424".i_xInterlock := FALSE;
       #"Conveyor 424"(i_xRun := TRUE,
                       ControlPanel := "General".Panel01,
                       q_xMotorOn => "Zne04 Conveyor 424",
                       Conveyor := "General"."Conveyor 424");
   END_REGION

   REGION "Conveyor 425"    
       #"Conveyor 425".i_xInterlock := FALSE;
       #"Conveyor 425"(i_xRun := TRUE,
                       ControlPanel := "General".Panel01,
                       q_xMotorOn => "Zne04 Conveyor 425",
                       Conveyor := "General"."Conveyor 425");
   END_REGION
END_FUNCTION_BLOCK

// folder: ZNE05

FUNCTION_BLOCK "Zne05"   // FB12, SCL
{ S7_Optimized_Access := 'TRUE' }
VERSION : 0.1
   VAR
      "Conveyor 500" : "Conveyor";
      "Conveyor 501" : "Conveyor";
      "Conveyor 502" : "Conveyor";
      "Pusher Zne05" : "Pusher";
      "Assembler Zne05" : "Assembler";
   END_VAR
BEGIN

   REGION "Conveyor 500"
       #"Conveyor 500".i_xInterlock := (NOT "General"."Assembler Zne05".ReadyToReceiveBase) AND "Sensor 500";
       #"Conveyor 500"(i_xRun := TRUE,
                       ControlPanel := "General".Panel01,
                       q_xMotorOn => "Zne05 Conveyor 500",
                       Conveyor := "General"."Conveyor 500");
   END_REGION

   REGION "Conveyor 501"
       #"Conveyor 501".i_xInterlock := FALSE;
       #"Conveyor 501"(i_xRun := TRUE,
                       ControlPanel := "General".Panel01,
                       q_xMotorOn => "Zne05 Conveyor 501",
                       Conveyor := "General"."Conveyor 501");
   END_REGION

   REGION "Conveyor 502"
       #"Conveyor 502".i_xInterlock := FALSE;
       #"Conveyor 502"(i_xRun := TRUE,
                       ControlPanel := "General".Panel01,
                       q_xMotorOn => "Zne05 Conveyor 502",
                       Conveyor := "General"."Conveyor 502");
   END_REGION

   REGION "Pusher Zne05"
       #"Pusher Zne05".RequestPusher := ("Vision Sensor 3 (Value)" <> "BlueBaseMaterial") AND ("Vision Sensor 3 (Value)" <> 0);
       #"Pusher Zne05"(Timer := T#500ms,
                       ControlPanel := "General".Panel01,
                       Pusher => "Zne05 Pusher");
   END_REGION

   REGION "Assembler"   
       "General"."Assembler Zne05".EnableSend := #"Conveyor 502".q_xMotorOn AND NOT "Sensor 502";
       #"Assembler Zne05"(LidClampClosed := "Zne04 Clamp Closed",
                          LidClampLimit := "Zne04 Clamp Limit",
                          BaseClampClosed := "Zne05 Clamp Closed",
                          BaseClampLimit := "Zne05 Clamp Limit",
                          PresenceLidConveyor := "Sensor 425",
                          PresenceBaseConveyor := "Sensor 501",
                          PresenceGrab := "Zne05 (Detected)",
                          MovingX := "Zne05 (Moving X)",
                          MovingZ := "Zne05 (Moving Z)",
                          ControlPanel := "General".Panel01,
                          LidClampClose => "Zne04 Clamp",
                          LidClampRise => "Zne04 Clamp Raise",
                          BaseClampClose => "Zne05 Clamp",
                          BaseClampRise => "Zne05 Clamp Raise",
                          AxisX => "Zne05 X",
                          AxisZ => "Zne05 Z",
                          Grab => "Zne05 (Grab)",
                          "St_ Assembler" := "General"."Assembler Zne05");
   END_REGION
END_FUNCTION_BLOCK

// folder: ZNE09

FUNCTION_BLOCK "Zne09"   // FB13, SCL
{ S7_Optimized_Access := 'TRUE' }
VERSION : 0.1
   VAR
      "Conveyor 920" : "Conveyor";
      "Conveyor 921" : "Conveyor";
      "Manipulator 1" : "Manipulator";
      "Conveyor 930" : "Conveyor";
      "Conveyor 931" : "Conveyor";
      "Manipulator 0" : "Manipulator";
      "Transfer Zne09" : "Transfer";
      "Conveyor 950" : "Conveyor";
      "Conveyor 951" : "Conveyor";
      Warehouse : "Warehouse";
      "Conveyor 952" : "Conveyor";
      "Conveyor 953" : "Conveyor";
      "tConveyor950 Interlock" : TOF_TIME;
   END_VAR
BEGIN


   REGION "Conveyor 920"    
       #"Conveyor 920"(i_xRun := "General"."Manipulator 1".ReadyToReceivePallet OR "General"."Manipulator 1".PalletFull,
                       ControlPanel := "General".Panel01,
                       q_xMotorOn => "Zne09 Conveyor 920",
                       Conveyor := "General"."Conveyor 920");
   END_REGION

   REGION "Manipulator 1"
       "General"."Manipulator 1".ContMax := 3;
       #"Manipulator 1"("Pallet Detected":="Sensor 920",
                        "Part Detected":="Sensor 302",
                        PresenceGrab:="Pick & Place 1 (Box Detected)",
                        "Actual Position X":="Pick & Place 1 X Position (V)",
                        "Actual Position Y":="Pick & Place 1 Y Position (V)",
                        "Actual Position Z":="Pick & Place 1 Z Position (V)",
                        ControlPanel:="General".Panel01,
                        "X Setpoint"=>"Pick & Place 1 X Set Point (V)",
                        "Y Setpoint"=>"Pick & Place 1 Y Set Point(V)",
                        "Z Setpoint"=>"Pick & Place 1 Z Set Point (V)",
                        Grab=>"Pick & Place 1 (Grab)",
                        Manipulator:="General"."Manipulator 1");
   END_REGION

   REGION "Conveyor 921"
       #"Conveyor 921".i_xInterlock := "Sensor 921" AND NOT "General".Transfer.ReadyToReceiveRight;
       #"Conveyor 921"(i_xRun := TRUE,
                       ControlPanel := "General".Panel01,
                       q_xMotorOn => "Zne09 Conveyor 921",
                       Conveyor := "General"."Conveyor 921");
   END_REGION

   REGION "Conveyor 930"    
       #"Conveyor 930"(i_xRun := "General"."Manipulator 0".ReadyToReceivePallet OR "General"."Manipulator 0".PalletFull,
                       ControlPanel := "General".Panel01,
                       q_xMotorOn => "Zne09 Conveyor 930",
                       Conveyor := "General"."Conveyor 930");
   END_REGION

   REGION "Manipulator 0"
       "General"."Manipulator 0".ContMax := 3;
       #"Manipulator 0"("Pallet Detected" := "Sensor 930",
                        "Part Detected" := "Sensor 502",
                        PresenceGrab := "Pick & Place 0 (Box Detected)",
                        "Actual Position X" := "Pick & Place 0 X Position (V)",
                        "Actual Position Y" := "Pick & Place 0 Y Position (V)",
                        "Actual Position Z" := "Pick & Place 0 Z Position (V)",
                        ControlPanel := "General".Panel01,
                        "X Setpoint" => "Pick & Place 0 X Set Point (V)",
                        "Y Setpoint" => "Pick & Place 0 Y Set Point(V)",
                        "Z Setpoint" => "Pick & Place 0 Z Set Point (V)",
                        Grab => "Pick & Place 0 (Grab)",
                        Manipulator := "General"."Manipulator 0");
   END_REGION

   REGION "Conveyor 931"
       #"Conveyor 931".i_xInterlock := "Sensor 931" AND NOT "General".Transfer.ReadyToReceiveLeft;
       #"Conveyor 931"(i_xRun := TRUE,
                       ControlPanel := "General".Panel01,
                       q_xMotorOn => "Zne09 Conveyor 931",
                       Conveyor := "General"."Conveyor 931");
   END_REGION

   REGION #"Transfer Zne09"
       "General".Transfer.EnableSend := "Sensor 950";
       "General".Transfer.RequestRight := "Sensor 921";
       "General".Transfer.RequestLeft := "Sensor 931";

       #"Transfer Zne09"(RightStop:="Sensor 922",
                         LeftStop:="Sensor 932",
                         ControlPanel:="General".Panel01,
                         "Chain Transfer Foward" =>"Zne09 Chain Transfer Foward",
                         "Chain Transfer Backward" =>"Zne09 Chain Transfer Backward",
                         "Chain Transfer Left" =>"Zne09 Chain Transfer Left",
                         "Chain Transfer Right" => "Zne09 Chain Transfer Right",
                         "Transfer":="General".Transfer);
   END_REGION

   REGION "Conveyor 950"    
       #"tConveyor950 Interlock"(IN:=NOT "Sensor 950" AND NOT "Sensor 951", PT:=t#2s);
       #"Conveyor 950"(i_xInterlock := #"tConveyor950 Interlock".Q,
                       i_xRun := TRUE,
                       ControlPanel := "General".Panel01,
                       q_xMotorOn => "Zne09 Conveyor 950",
                       Conveyor := "General"."Conveyor 950");
   END_REGION

   REGION "Conveyor 951"
       #"Conveyor 951"(i_xInterlock:=NOT "Sensor 951",
                       i_xRun:=TRUE,
                       ControlPanel:="General".Panel01,
                       q_xMotorOn=>"Zne09 Conveyor 951",
                       Conveyor:="General"."Conveyor 951");
   END_REGION

   REGION Wirehouse    
       "General".Warehouse.xSensorEntrada := NOT "Sensor 951";
       "General".Warehouse.xSensorSaida := NOT "Sensor 952";

       #Warehouse(i_xAtLeft:="AtLeft",
                  i_xAtRight:="AtRight",
                  i_xAtMiddle:="AtCenter",
                  i_xMovingZ:="MovingZ",
                  i_xMovingX:="MovingX",
                  ControlPanel:="General".Panel01,
                  q_xForksLeft=>"ForksLeft",
                  q_xForksRight=>"Forks RIght",
                  q_xLift=>"Lift",
                  q_dTargetPosition=> "Zne09 Stacker Target Position",
                  Warehouse:="General".Warehouse);
   END_REGION

   REGION #"Conveyor 952"
       #"Conveyor 952"(i_xRun := TRUE,
                       ControlPanel := "General".Panel01,
                       q_xMotorOn => "Zne09 Conveyor 952",
                       Conveyor := "General"."Conveyor 952");
   END_REGION

   REGION #"Conveyor 953"
       #"Conveyor 953"(i_xRun := TRUE,
                       ControlPanel := "General".Panel01,
                       q_xMotorOn => "Zne09 Conveyor 953",
                       Conveyor := "General"."Conveyor 953");
   END_REGION
END_FUNCTION_BLOCK

FUNCTION "Receita" : Void   // FC3, SCL
{ S7_Optimized_Access := 'TRUE' }
VERSION : 0.1
BEGIN
   REGION "Manipulator" 1       
       // HOME
       "General"."Manipulator 1".Coordinates[0]."Axis X" := 11664;
       "General"."Manipulator 1".Coordinates[0]."Axis Y" := 10368;
       "General"."Manipulator 1".Coordinates[0]."Axis Z" := 1000;

       // PREPICK
       "General"."Manipulator 1".Coordinates[1]."Axis X" := 19872;
       "General"."Manipulator 1".Coordinates[1]."Axis Y" := 14688;
       "General"."Manipulator 1".Coordinates[1]."Axis Z" := 1000;

       // PICK
       "General"."Manipulator 1".Coordinates[2]."Axis X" := 19872;
       "General"."Manipulator 1".Coordinates[2]."Axis Y" := 14688;
       "General"."Manipulator 1".Coordinates[2]."Axis Z" := 21607;

       // POSPICK
       "General"."Manipulator 1".Coordinates[3]."Axis X" := 19872;
       "General"."Manipulator 1".Coordinates[3]."Axis Y" := 14688;
       "General"."Manipulator 1".Coordinates[3]."Axis Z" := 10000;

       // PREDROP
       "General"."Manipulator 1".Coordinates[4]."Axis X" := 6912;
       "General"."Manipulator 1".Coordinates[4]."Axis Y" := 14688;
       "General"."Manipulator 1".Coordinates[4]."Axis Z" := 10000;

       // DROP
       "General"."Manipulator 1".Coordinates[5]."Axis X" := 6912;
       "General"."Manipulator 1".Coordinates[5]."Axis Y" := 14688;
       "General"."Manipulator 1".Coordinates[5]."Axis Z" := 27648 - ("General"."Manipulator 1".ContActual * 2000);

       // POSDROP
       "General"."Manipulator 1".Coordinates[6]."Axis X" := 6912;
       "General"."Manipulator 1".Coordinates[6]."Axis Y" := 14688;
       "General"."Manipulator 1".Coordinates[6]."Axis Z" := 15124;
   END_REGION

   REGION "Manipulator" 0       
       // HOME
       "General"."Manipulator 0".Coordinates[0]."Axis X" := 11664;
       "General"."Manipulator 0".Coordinates[0]."Axis Y" := 10368;
       "General"."Manipulator 0".Coordinates[0]."Axis Z" := 1000;

       // PREPICK
       "General"."Manipulator 0".Coordinates[1]."Axis X" := 19872;
       "General"."Manipulator 0".Coordinates[1]."Axis Y" := 14688;
       "General"."Manipulator 0".Coordinates[1]."Axis Z" := 1000;

       // PICK
       "General"."Manipulator 0".Coordinates[2]."Axis X" := 19872;
       "General"."Manipulator 0".Coordinates[2]."Axis Y" := 14688;
       "General"."Manipulator 0".Coordinates[2]."Axis Z" := 21607;

       // POSPICK
       "General"."Manipulator 0".Coordinates[3]."Axis X" := 19872;
       "General"."Manipulator 0".Coordinates[3]."Axis Y" := 14688;
       "General"."Manipulator 0".Coordinates[3]."Axis Z" := 10000;

       // PREDROP
       "General"."Manipulator 0".Coordinates[4]."Axis X" := 6912;
       "General"."Manipulator 0".Coordinates[4]."Axis Y" := 14688;
       "General"."Manipulator 0".Coordinates[4]."Axis Z" := 10000;

       // DROP
       "General"."Manipulator 0".Coordinates[5]."Axis X" := 6912;
       "General"."Manipulator 0".Coordinates[5]."Axis Y" := 14688;
       "General"."Manipulator 0".Coordinates[5]."Axis Z" := 27648 - ("General"."Manipulator 0".ContActual * 2000);

       // POSDROP
       "General"."Manipulator 0".Coordinates[6]."Axis X" := 6912;
       "General"."Manipulator 0".Coordinates[6]."Axis Y" := 14688;
       "General"."Manipulator 0".Coordinates[6]."Axis Z" := 15124;
   END_REGION
END_FUNCTION